LIN {X 0,Y 162.766,Z 348.566,A -85,B 0,C 180,E1 -23650.117,E2 -23650.117} C_VEL
LIN {X 0,Y 165.298,Z 338.62,A -85,B 0,C 180,E1 -23653.005,E2 -23653.005} C_VEL
LIN {X 0,Y 166.712,Z 332.788,A -85,B 0,C 180,E1 -23654.411,E2 -23654.411} C_VEL
LIN {X 0,Y 165.838,Z 322.83,A -85,B 0,C 180,E1 -23656.834,E2 -23656.834} C_VEL
LIN {X 0,Y 164.302,Z 311.523,A -85,B 0,C 180,E1 -23659.215,E2 -23659.215} C_VEL
LIN {X 0,Y 162.119,Z 300.27,A -85,B 0,C 180,E1 -23661.273,E2 -23661.273} C_VEL
LIN {X 0,Y 158.794,Z 286.809,A -85,B 0,C 180,E1 -23663.369,E2 -23663.369} C_VEL
LIN {X 0,Y 157.682,Z 283.839,A -85,B 0,C 180,E1 -23663.924,E2 -23663.924} C_VEL
LIN {X 0,Y 158.248,Z 283.771,A -85,B 0,C 180,E1 -23670,E2 -23670} C_VEL
LIN {X 0,Y 157.816,Z 283.83,A -85,B 0,C 180,E1 -23677.678,E2 -23677.678} C_VEL
LIN {X 0,Y 157.697,Z 283.837,A -85,B 0,C 180,E1 -23681.363,E2 -23681.363} C_VEL
LIN {X 0,Y 157.479,Z 283.868,A -85,B 0,C 180,E1 -23685.532,E2 -23685.532} C_VEL
LIN {X 0,Y 157.407,Z 283.876,A -85,B 0,C 180,E1 -23690.928,E2 -23690.928} C_VEL
LIN {X 0,Y 157.306,Z 283.879,A -85,B 0,C 180,E1 -23696.686,E2 -23696.686} C_VEL
LIN {X 0,Y 157.269,Z 283.893,A -85,B 0,C 180,E1 -23702.429,E2 -23702.429} C_VEL
LIN {X 0,Y 157.318,Z 283.886,A -85,B 0,C 180,E1 -23706.479,E2 -23706.479} C_VEL
LIN {X 0,Y 157.288,Z 283.866,A -85,B 0,C 180,E1 -23712.085,E2 -23712.085} C_VEL
LIN {X 0,Y 157.304,Z 283.881,A -85,B 0,C 180,E1 -23715.63,E2 -23715.63} C_VEL
LIN {X 0,Y 157.284,Z 283.893,A -85,B 0,C 180,E1 -23721.28,E2 -23721.28} C_VEL
LIN {X 0,Y 157.289,Z 283.885,A -85,B 0,C 180,E1 -23724.493,E2 -23724.493} C_VEL
LIN {X 0,Y 157.289,Z 283.864,A -85,B 0,C 180,E1 -23728.098,E2 -23728.098} C_VEL
LIN {X 0,Y 157.317,Z 283.878,A -85,B 0,C 180,E1 -23733.469,E2 -23733.469} C_VEL
LIN {X 0,Y 157.39,Z 283.878,A -85,B 0,C 180,E1 -23739.671,E2 -23739.671} C_VEL
LIN {X 0,Y 157.438,Z 283.857,A -85,B 0,C 180,E1 -23744.468,E2 -23744.468} C_VEL
LIN {X 0,Y 157.686,Z 283.82,A -85,B 0,C 180,E1 -23749.734,E2 -23749.734} C_VEL
LIN {X 0,Y 157.765,Z 283.822,A -85,B 0,C 180,E1 -23752.323,E2 -23752.323} C_VEL
LIN {X 0,Y 158.255,Z 283.768,A -85,B 0,C 180,E1 -23760.003,E2 -23760.003} C_VEL
LIN {X 0,Y 157.803,Z 283.815,A -85,B 0,C 180,E1 -23767.681,E2 -23767.681} C_VEL
LIN {X 0,Y 157.681,Z 283.842,A -85,B 0,C 180,E1 -23771.319,E2 -23771.319} C_VEL
LIN {X 0,Y 157.478,Z 283.864,A -85,B 0,C 180,E1 -23775.535,E2 -23775.535} C_VEL
LIN {X 0,Y 157.372,Z 283.876,A -85,B 0,C 180,E1 -23780.936,E2 -23780.936} C_VEL
LIN {X 0,Y 157.317,Z 283.884,A -85,B 0,C 180,E1 -23786.687,E2 -23786.687} C_VEL
LIN {X 0,Y 157.278,Z 283.896,A -85,B 0,C 180,E1 -23792.43,E2 -23792.43} C_VEL
LIN {X 0,Y 157.273,Z 283.892,A -85,B 0,C 180,E1 -23796.452,E2 -23796.452} C_VEL
LIN {X 0,Y 157.389,Z 283.892,A -85,B 0,C 180,E1 -23801.622,E2 -23801.622} C_VEL
LIN {X 0,Y 157.799,Z 286.274,A -85,B 0,C 180,E1 -23805.451,E2 -23805.451} C_VEL
LIN {X 0,Y 158.208,Z 288.611,A -85,B 0,C 180,E1 -23809.045,E2 -23809.045} C_VEL
LIN {X 0,Y 158.559,Z 290.868,A -85,B 0,C 180,E1 -23812.25,E2 -23812.25} C_VEL
LIN {X 0,Y 161.072,Z 302.499,A -85,B 0,C 180,E1 -23813.8,E2 -23813.8} C_VEL
LIN {X 0,Y 162.819,Z 314.796,A -85,B 0,C 180,E1 -23815.699,E2 -23815.699} C_VEL
LIN {X 0,Y 164.125,Z 327.048,A -85,B 0,C 180,E1 -23818.002,E2 -23818.002} C_VEL
LIN {X 0,Y 164.669,Z 338.78,A -85,B 0,C 180,E1 -23820.606,E2 -23820.606} C_VEL
LIN {X 0,Y 164.749,Z 346.799,A -85,B 0,C 180,E1 -23822.705,E2 -23822.705} C_VEL
LIN {X 0,Y 162.212,Z 356.942,A -85,B 0,C 180,E1 -23825.614,E2 -23825.614} C_VEL
LIN {X 0,Y 159.951,Z 365.602,A -85,B 0,C 180,E1 -23828.747,E2 -23828.747} C_VEL
LIN {X 0,Y 157.78,Z 373.82,A -85,B 0,C 180,E1 -23832.502,E2 -23832.502} C_VEL
LIN {X 0,Y 156.445,Z 379.436,A -85,B 0,C 180,E1 -23835.695,E2 -23835.695} C_VEL
LIN {X 0,Y 155.464,Z 384.917,A -85,B 0,C 180,E1 -23839.582,E2 -23839.582} C_VEL
LIN {X 0,Y 154.93,Z 389.177,A -85,B 0,C 180,E1 -23843.488,E2 -23843.488} C_VEL
LIN {X 0,Y 154.782,Z 392.343,A -85,B 0,C 180,E1 -23847.397,E2 -23847.397} C_VEL
LIN {X 0,Y 154.902,Z 393.899,A -85,B 0,C 180,E1 -23850,E2 -23850} C_VEL
LIN {X 0,Y 154.782,Z 395.024,A -85,B 0,C 180,E1 -23852.602,E2 -23852.602} C_VEL
LIN {X 0,Y 154.786,Z 395.727,A -85,B 0,C 180,E1 -23855.21,E2 -23855.21} C_VEL
LIN {X 0,Y 155.452,Z 395.975,A -85,B 0,C 180,E1 -23860.418,E2 -23860.418} C_VEL
LIN {X 0,Y 157.219,Z 394.762,A -85,B 0,C 180,E1 -23865.557,E2 -23865.557} C_VEL
LIN {X 0,Y 158.527,Z 393.574,A -85,B 0,C 180,E1 -23868.078,E2 -23868.078} C_VEL
LIN {X 0,Y 162.36,Z 390.018,A -85,B 0,C 180,E1 -23872.927,E2 -23872.927} C_VEL
LIN {X 0,Y 165.867,Z 386.263,A -85,B 0,C 180,E1 -23876.416,E2 -23876.416} C_VEL
LIN {X 0,Y 169.84,Z 381.521,A -85,B 0,C 180,E1 -23879.772,E2 -23879.772} C_VEL
LIN {X 0,Y 175.416,Z 374.551,A -85,B 0,C 180,E1 -23883.427,E2 -23883.427} C_VEL
LIN {X 0,Y 180.894,Z 367.066,A -85,B 0,C 180,E1 -23886.332,E2 -23886.332} C_VEL
LIN {X 0,Y 182.456,Z 364.28,A -85,B 0,C 180,E1 -23887.348,E2 -23887.348} C_VEL
LIN {X 0,Y 184.669,Z 357.993,A -85,B 0,C 180,E1 -23889.824,E2 -23889.824} C_VEL
LIN {X 0,Y 185.443,Z 355.091,A -85,B 0,C 180,E1 -23890.981,E2 -23890.981} C_VEL
LIN {X 0,Y 185.682,Z 351.795,A -85,B 0,C 180,E1 -23892.493,E2 -23892.493} C_VEL
LIN {X 0,Y 184.975,Z 349.138,A -85,B 0,C 180,E1 -23894.125,E2 -23894.125} C_VEL
LIN {X 0,Y 181.89,Z 343.339,A -85,B 0,C 180,E1 -23898.777,E2 -23898.777} C_VEL
LIN {X 0,Y 181.489,Z 341.7,A -85,B 0,C 180,E1 -23899.951,E2 -23899.951} C_VEL
LIN {X 0,Y 180.807,Z 337.52,A -85,B 0,C 180,E1 -23902.909,E2 -23902.909} C_VEL
LIN {X 0,Y 180.236,Z 335.055,A -85,B 0,C 180,E1 -23904.969,E2 -23904.969} C_VEL
LIN {X 0,Y 179.745,Z 332.311,A -85,B 0,C 180,E1 -23907.505,E2 -23907.505} C_VEL
LIN {X 0,Y 178.614,Z 327.494,A -85,B 0,C 180,E1 -23914.819,E2 -23914.819} C_VEL
LIN {X 0,Y 178.644,Z 326.719,A -85,B 0,C 180,E1 -23916.831,E2 -23916.831} C_VEL
LIN {X 0,Y 178.742,Z 326.277,A -85,B 0,C 180,E1 -23919.273,E2 -23919.273} C_VEL
LIN {X 0,Y 178.794,Z 326.661,A -85,B 0,C 180,E1 -23921.669,E2 -23921.669} C_VEL
LIN {X 0,Y 180.094,Z 329.764,A -85,B 0,C 180,E1 -23928.746,E2 -23928.746} C_VEL
LIN {X 0,Y 181.755,Z 335.002,A -85,B 0,C 180,E1 -23934.45,E2 -23934.45} C_VEL
LIN {X 0,Y 182.467,Z 339.478,A -85,B 0,C 180,E1 -23937.79,E2 -23937.79} C_VEL
LIN {X 0,Y 182.834,Z 344.048,A -85,B 0,C 180,E1 -23940.659,E2 -23940.659} C_VEL
LIN {X 0,Y 182.159,Z 350.277,A -85,B 0,C 180,E1 -23943.869,E2 -23943.869} C_VEL
LIN {X 0,Y 180.695,Z 356.16,A -85,B 0,C 180,E1 -23946.698,E2 -23946.698} C_VEL
LIN {X 0,Y 179.669,Z 358.308,A -85,B 0,C 180,E1 -23947.574,E2 -23947.574} C_VEL
LIN {X 0,Y 174.172,Z 365.633,A -85,B 0,C 180,E1 -23950.28,E2 -23950.28} C_VEL
LIN {X 0,Y 168.006,Z 372.913,A -85,B 0,C 180,E1 -23953.83,E2 -23953.83} C_VEL
LIN {X 0,Y 162.389,Z 378.767,A -85,B 0,C 180,E1 -23957.804,E2 -23957.804} C_VEL
LIN {X 0,Y 157.176,Z 383.446,A -85,B 0,C 180,E1 -23962.497,E2 -23962.497} C_VEL
LIN {X 0,Y 153.192,Z 386.436,A -85,B 0,C 180,E1 -23967.304,E2 -23967.304} C_VEL
LIN {X 0,Y 150.147,Z 387.993,A -85,B 0,C 180,E1 -23972.594,E2 -23972.594} C_VEL
LIN {X 0,Y 148.174,Z 388.041,A -85,B 0,C 180,E1 -23978.064,E2 -23978.064} C_VEL
LIN {X 0,Y 147.408,Z 387.123,A -85,B 0,C 180,E1 -23981.868,E2 -23981.868} C_VEL
LIN {X 0,Y 147.139,Z 385.428,A -85,B 0,C 180,E1 -23985.758,E2 -23985.758} C_VEL
LIN {X 0,Y 147.295,Z 382.83,A -85,B 0,C 180,E1 -23989.761,E2 -23989.761} C_VEL
LIN {X 0,Y 147.963,Z 379.18,A -85,B 0,C 180,E1 -23993.843,E2 -23993.843} C_VEL
LIN {X 0,Y 149.28,Z 373.176,A -85,B 0,C 180,E1 -23998.812,E2 -23998.812} C_VEL
LIN {X 0,Y 151.04,Z 366.254,A -85,B 0,C 180,E1 -24003.15,E2 -24003.15} C_VEL
LIN {X 0,Y 153.366,Z 357.835,A -85,B 0,C 180,E1 -24007.228,E2 -24007.228} C_VEL
LIN {X 0,Y 155.725,Z 349.243,A -85,B 0,C 180,E1 -24010.534,E2 -24010.534} C_VEL
LIN {X 0,Y 158.317,Z 339.375,A -85,B 0,C 180,E1 -24013.562,E2 -24013.562} C_VEL
LIN {X 0,Y 159.876,Z 332.712,A -85,B 0,C 180,E1 -24015.248,E2 -24015.248} C_VEL
LIN {X 0,Y 158.746,Z 321.108,A -85,B 0,C 180,E1 -24018.185,E2 -24018.185} C_VEL
LIN {X 0,Y 157.013,Z 309.073,A -85,B 0,C 180,E1 -24020.76,E2 -24020.76} C_VEL
LIN {X 0,Y 154.341,Z 296.343,A -85,B 0,C 180,E1 -24023.135,E2 -24023.135} C_VEL
LIN {X 0,Y 152.56,Z 289.599,A -85,B 0,C 180,E1 -24024.258,E2 -24024.258} C_VEL
LIN {X 0,Y 150.695,Z 285.026,A -85,B 0,C 180,E1 -24025.068,E2 -24025.068} C_VEL
LIN {X 0,Y 150.666,Z 284.718,A -85,B 0,C 180,E1 -24025.318,E2 -24025.318} C_VEL
LIN {X 0,Y 151.208,Z 284.648,A -85,B 0,C 180,E1 -24030,E2 -24030} C_VEL
LIN {X 0,Y 150.754,Z 284.71,A -85,B 0,C 180,E1 -24038.04,E2 -24038.04} C_VEL
LIN {X 0,Y 150.626,Z 284.718,A -85,B 0,C 180,E1 -24041.546,E2 -24041.546} C_VEL
LIN {X 0,Y 150.388,Z 284.747,A -85,B 0,C 180,E1 -24046.284,E2 -24046.284} C_VEL
LIN {X 0,Y 150.382,Z 284.751,A -85,B 0,C 180,E1 -24050.832,E2 -24050.832} C_VEL
LIN {X 0,Y 150.236,Z 284.755,A -85,B 0,C 180,E1 -24057.283,E2 -24057.283} C_VEL
LIN {X 0,Y 150.21,Z 284.773,A -85,B 0,C 180,E1 -24062.636,E2 -24062.636} C_VEL
LIN {X 0,Y 150.229,Z 284.766,A -85,B 0,C 180,E1 -24067.457,E2 -24067.457} C_VEL
LIN {X 0,Y 150.229,Z 284.745,A -85,B 0,C 180,E1 -24071.544,E2 -24071.544} C_VEL
LIN {X 0,Y 150.254,Z 284.757,A -85,B 0,C 180,E1 -24075.449,E2 -24075.449} C_VEL
LIN {X 0,Y 150.229,Z 284.771,A -85,B 0,C 180,E1 -24079.089,E2 -24079.089} C_VEL
LIN {X 0,Y 150.233,Z 284.769,A -85,B 0,C 180,E1 -24082.68,E2 -24082.68} C_VEL
LIN {X 0,Y 150.213,Z 284.748,A -85,B 0,C 180,E1 -24087.368,E2 -24087.368} C_VEL
LIN {X 0,Y 150.239,Z 284.754,A -85,B 0,C 180,E1 -24092.721,E2 -24092.721} C_VEL
LIN {X 0,Y 150.347,Z 284.756,A -85,B 0,C 180,E1 -24099.211,E2 -24099.211} C_VEL
LIN {X 0,Y 150.349,Z 284.745,A -85,B 0,C 180,E1 -24103.715,E2 -24103.715} C_VEL
LIN {X 0,Y 150.606,Z 284.696,A -85,B 0,C 180,E1 -24109.245,E2 -24109.245} C_VEL
LIN {X 0,Y 150.702,Z 284.7,A -85,B 0,C 180,E1 -24111.961,E2 -24111.961} C_VEL
LIN {X 0,Y 151.216,Z 284.644,A -85,B 0,C 180,E1 -24120.003,E2 -24120.003} C_VEL
LIN {X 0,Y 150.739,Z 284.696,A -85,B 0,C 180,E1 -24128.044,E2 -24128.044} C_VEL
LIN {X 0,Y 150.612,Z 284.723,A -85,B 0,C 180,E1 -24131.504,E2 -24131.504} C_VEL
LIN {X 0,Y 150.382,Z 284.743,A -85,B 0,C 180,E1 -24136.288,E2 -24136.288} C_VEL
LIN {X 0,Y 150.353,Z 284.75,A -85,B 0,C 180,E1 -24140.795,E2 -24140.795} C_VEL
LIN {X 0,Y 150.247,Z 284.762,A -85,B 0,C 180,E1 -24147.285,E2 -24147.285} C_VEL
LIN {X 0,Y 150.218,Z 284.776,A -85,B 0,C 180,E1 -24152.635,E2 -24152.635} C_VEL
LIN {X 0,Y 150.184,Z 284.779,A -85,B 0,C 180,E1 -24157.474,E2 -24157.474} C_VEL
LIN {X 0,Y 150.378,Z 284.841,A -85,B 0,C 180,E1 -24161.603,E2 -24161.603} C_VEL
LIN {X 0,Y 150.77,Z 287.258,A -85,B 0,C 180,E1 -24165.637,E2 -24165.637} C_VEL
LIN {X 0,Y 151.334,Z 290.659,A -85,B 0,C 180,E1 -24170.886,E2 -24170.886} C_VEL
LIN {X 0,Y 153.685,Z 298.998,A -85,B 0,C 180,E1 -24172.13,E2 -24172.13} C_VEL
LIN {X 0,Y 155.558,Z 311.145,A -85,B 0,C 180,E1 -24174.032,E2 -24174.032} C_VEL
LIN {X 0,Y 157.072,Z 324.55,A -85,B 0,C 180,E1 -24176.557,E2 -24176.557} C_VEL
LIN {X 0,Y 157.706,Z 335.061,A -85,B 0,C 180,E1 -24178.909,E2 -24178.909} C_VEL
LIN {X 0,Y 157.848,Z 345.901,A -85,B 0,C 180,E1 -24181.767,E2 -24181.767} C_VEL
LIN {X 0,Y 157.329,Z 349.398,A -85,B 0,C 180,E1 -24182.75,E2 -24182.75} C_VEL
LIN {X 0,Y 154.633,Z 359.142,A -85,B 0,C 180,E1 -24185.855,E2 -24185.855} C_VEL
LIN {X 0,Y 152.479,Z 367.199,A -85,B 0,C 180,E1 -24189.071,E2 -24189.071} C_VEL
LIN {X 0,Y 150.344,Z 375.101,A -85,B 0,C 180,E1 -24193.012,E2 -24193.012} C_VEL
LIN {X 0,Y 149.099,Z 380.453,A -85,B 0,C 180,E1 -24196.368,E2 -24196.368} C_VEL
LIN {X 0,Y 148.219,Z 385.687,A -85,B 0,C 180,E1 -24200.447,E2 -24200.447} C_VEL
LIN {X 0,Y 147.775,Z 389.713,A -85,B 0,C 180,E1 -24204.542,E2 -24204.542} C_VEL
LIN {X 0,Y 147.695,Z 392.183,A -85,B 0,C 180,E1 -24207.89,E2 -24207.89} C_VEL
LIN {X 0,Y 147.809,Z 393.41,A -85,B 0,C 180,E1 -24210,E2 -24210} C_VEL
LIN {X 0,Y 147.701,Z 394.601,A -85,B 0,C 180,E1 -24212.727,E2 -24212.727} C_VEL
LIN {X 0,Y 147.709,Z 395.398,A -85,B 0,C 180,E1 -24215.46,E2 -24215.46} C_VEL
LIN {X 0,Y 147.947,Z 395.797,A -85,B 0,C 180,E1 -24218.193,E2 -24218.193} C_VEL
LIN {X 0,Y 149.258,Z 395.448,A -85,B 0,C 180,E1 -24223.616,E2 -24223.616} C_VEL
LIN {X 0,Y 151.779,Z 393.647,A -85,B 0,C 180,E1 -24228.912,E2 -24228.912} C_VEL
LIN {X 0,Y 153.631,Z 392.168,A -85,B 0,C 180,E1 -24231.466,E2 -24231.466} C_VEL
LIN {X 0,Y 158.258,Z 387.996,A -85,B 0,C 180,E1 -24236.364,E2 -24236.364} C_VEL
LIN {X 0,Y 162.767,Z 383.216,A -85,B 0,C 180,E1 -24240.276,E2 -24240.276} C_VEL
LIN {X 0,Y 167.85,Z 377.486,A -85,B 0,C 180,E1 -24243.695,E2 -24243.695} C_VEL
LIN {X 0,Y 173.286,Z 370.738,A -85,B 0,C 180,E1 -24246.741,E2 -24246.741} C_VEL
LIN {X 0,Y 176.227,Z 366.828,A -85,B 0,C 180,E1 -24248.18,E2 -24248.18} C_VEL
LIN {X 0,Y 178.837,Z 360.757,A -85,B 0,C 180,E1 -24250.756,E2 -24250.756} C_VEL
LIN {X 0,Y 180.785,Z 353.995,A -85,B 0,C 180,E1 -24253.63,E2 -24253.63} C_VEL
LIN {X 0,Y 181.779,Z 348.847,A -85,B 0,C 180,E1 -24255.896,E2 -24255.896} C_VEL
LIN {X 0,Y 181.866,Z 345.381,A -85,B 0,C 180,E1 -24257.706,E2 -24257.706} C_VEL
LIN {X 0,Y 181.489,Z 341.7,A -85,B 0,C 180,E1 -24259.951,E2 -24259.951} C_VEL
LIN {X 0,Y 180.704,Z 339.737,A -85,B 0,C 180,E1 -24261.691,E2 -24261.691} C_VEL
LIN {X 0,Y 179.33,Z 338.667,A -85,B 0,C 180,E1 -24263.499,E2 -24263.499} C_VEL
LIN {X 0,Y 175.537,Z 337.281,A -85,B 0,C 180,E1 -24268.542,E2 -24268.542} C_VEL
LIN {X 0,Y 175.12,Z 336.621,A -85,B 0,C 180,E1 -24269.837,E2 -24269.837} C_VEL
LIN {X 0,Y 174.769,Z 334.192,A -85,B 0,C 180,E1 -24273.744,E2 -24273.744} C_VEL
LIN {X 0,Y 174.924,Z 332.649,A -85,B 0,C 180,E1 -24277.527,E2 -24277.527} C_VEL
LIN {X 0,Y 174.99,Z 332.407,A -85,B 0,C 180,E1 -24278.807,E2 -24278.807} C_VEL
LIN {X 0,Y 175.063,Z 332.617,A -85,B 0,C 180,E1 -24281.264,E2 -24281.264} C_VEL
LIN {X 0,Y 175.996,Z 335.511,A -85,B 0,C 180,E1 -24288.48,E2 -24288.48} C_VEL
LIN {X 0,Y 176.957,Z 339.379,A -85,B 0,C 180,E1 -24293.154,E2 -24293.154} C_VEL
LIN {X 0,Y 177.5,Z 343.407,A -85,B 0,C 180,E1 -24296.592,E2 -24296.592} C_VEL
LIN {X 0,Y 177.562,Z 348.314,A -85,B 0,C 180,E1 -24299.997,E2 -24299.997} C_VEL
LIN {X 0,Y 176.637,Z 353.41,A -85,B 0,C 180,E1 -24302.849,E2 -24302.849} C_VEL
LIN {X 0,Y 174.875,Z 359.006,A -85,B 0,C 180,E1 -24305.764,E2 -24305.764} C_VEL
LIN {X 0,Y 168.913,Z 366.651,A -85,B 0,C 180,E1 -24308.725,E2 -24308.725} C_VEL
LIN {X 0,Y 162.138,Z 374.054,A -85,B 0,C 180,E1 -24312.514,E2 -24312.514} C_VEL
LIN {X 0,Y 156.233,Z 379.619,A -85,B 0,C 180,E1 -24316.572,E2 -24316.572} C_VEL
LIN {X 0,Y 150.852,Z 384.044,A -85,B 0,C 180,E1 -24321.291,E2 -24321.291} C_VEL
LIN {X 0,Y 147.222,Z 386.501,A -85,B 0,C 180,E1 -24325.441,E2 -24325.441} C_VEL
LIN {X 0,Y 144.751,Z 387.774,A -85,B 0,C 180,E1 -24329.083,E2 -24329.083} C_VEL
LIN {X 0,Y 142.717,Z 388.396,A -85,B 0,C 180,E1 -24333.162,E2 -24333.162} C_VEL
LIN {X 0,Y 141.269,Z 388.228,A -85,B 0,C 180,E1 -24337.254,E2 -24337.254} C_VEL
LIN {X 0,Y 140.381,Z 387.25,A -85,B 0,C 180,E1 -24341.329,E2 -24341.329} C_VEL
LIN {X 0,Y 140.06,Z 385.51,A -85,B 0,C 180,E1 -24345.374,E2 -24345.374} C_VEL
LIN {X 0,Y 140.156,Z 383.054,A -85,B 0,C 180,E1 -24349.318,E2 -24349.318} C_VEL
LIN {X 0,Y 140.693,Z 379.862,A -85,B 0,C 180,E1 -24353.172,E2 -24353.172} C_VEL
LIN {X 0,Y 141.702,Z 375.212,A -85,B 0,C 180,E1 -24357.467,E2 -24357.467} C_VEL
LIN {X 0,Y 143.303,Z 368.887,A -85,B 0,C 180,E1 -24361.971,E2 -24361.971} C_VEL
LIN {X 0,Y 145.594,Z 360.66,A -85,B 0,C 180,E1 -24366.504,E2 -24366.504} C_VEL
LIN {X 0,Y 148.102,Z 351.955,A -85,B 0,C 180,E1 -24370.239,E2 -24370.239} C_VEL
LIN {X 0,Y 151.029,Z 341.386,A -85,B 0,C 180,E1 -24373.788,E2 -24373.788} C_VEL
LIN {X 0,Y 152.807,Z 334.817,A -85,B 0,C 180,E1 -24375.586,E2 -24375.586} C_VEL
LIN {X 0,Y 152.839,Z 330.773,A -85,B 0,C 180,E1 -24376.709,E2 -24376.709} C_VEL
LIN {X 0,Y 151.648,Z 319.16,A -85,B 0,C 180,E1 -24379.689,E2 -24379.689} C_VEL
LIN {X 0,Y 150.15,Z 309.08,A -85,B 0,C 180,E1 -24381.928,E2 -24381.928} C_VEL
LIN {X 0,Y 147.75,Z 297.311,A -85,B 0,C 180,E1 -24384.225,E2 -24384.225} C_VEL
LIN {X 0,Y 146.372,Z 292.363,A -85,B 0,C 180,E1 -24385.137,E2 -24385.137} C_VEL
LIN {X 0,Y 143.867,Z 286.452,A -85,B 0,C 180,E1 -24386.324,E2 -24386.324} C_VEL
LIN {X 0,Y 143.73,Z 285.58,A -85,B 0,C 180,E1 -24386.496,E2 -24386.496} C_VEL
LIN {X 0,Y 144.166,Z 285.525,A -85,B 0,C 180,E1 -24390,E2 -24390} C_VEL
LIN {X 0,Y 143.676,Z 285.59,A -85,B 0,C 180,E1 -24398.439,E2 -24398.439} C_VEL
LIN {X 0,Y 143.563,Z 285.599,A -85,B 0,C 180,E1 -24401.759,E2 -24401.759} C_VEL
LIN {X 0,Y 143.326,Z 285.623,A -85,B 0,C 180,E1 -24407.11,E2 -24407.11} C_VEL
LIN {X 0,Y 143.303,Z 285.633,A -85,B 0,C 180,E1 -24411.291,E2 -24411.291} C_VEL
LIN {X 0,Y 143.182,Z 285.632,A -85,B 0,C 180,E1 -24417.938,E2 -24417.938} C_VEL
LIN {X 0,Y 143.161,Z 285.652,A -85,B 0,C 180,E1 -24423.437,E2 -24423.437} C_VEL
LIN {X 0,Y 143.122,Z 285.639,A -85,B 0,C 180,E1 -24429.67,E2 -24429.67} C_VEL
LIN {X 0,Y 143.161,Z 285.628,A -85,B 0,C 180,E1 -24433.415,E2 -24433.415} C_VEL
LIN {X 0,Y 143.156,Z 285.649,A -85,B 0,C 180,E1 -24437.425,E2 -24437.425} C_VEL
LIN {X 0,Y 143.137,Z 285.653,A -85,B 0,C 180,E1 -24441.775,E2 -24441.775} C_VEL
LIN {X 0,Y 143.18,Z 285.623,A -85,B 0,C 180,E1 -24447.325,E2 -24447.325} C_VEL
LIN {X 0,Y 143.185,Z 285.63,A -85,B 0,C 180,E1 -24452.066,E2 -24452.066} C_VEL
LIN {X 0,Y 143.273,Z 285.639,A -85,B 0,C 180,E1 -24458.749,E2 -24458.749} C_VEL
LIN {X 0,Y 143.292,Z 285.625,A -85,B 0,C 180,E1 -24462.889,E2 -24462.889} C_VEL
LIN {X 0,Y 143.532,Z 285.572,A -85,B 0,C 180,E1 -24468.709,E2 -24468.709} C_VEL
LIN {X 0,Y 143.623,Z 285.581,A -85,B 0,C 180,E1 -24471.562,E2 -24471.562} C_VEL
LIN {X 0,Y 144.175,Z 285.521,A -85,B 0,C 180,E1 -24480.003,E2 -24480.003} C_VEL
LIN {X 0,Y 143.66,Z 285.58,A -85,B 0,C 180,E1 -24488.443,E2 -24488.443} C_VEL
LIN {X 0,Y 143.549,Z 285.604,A -85,B 0,C 180,E1 -24491.716,E2 -24491.716} C_VEL
LIN {X 0,Y 143.317,Z 285.619,A -85,B 0,C 180,E1 -24497.115,E2 -24497.115} C_VEL
LIN {X 0,Y 143.279,Z 285.632,A -85,B 0,C 180,E1 -24501.257,E2 -24501.257} C_VEL
LIN {X 0,Y 143.193,Z 285.639,A -85,B 0,C 180,E1 -24507.94,E2 -24507.94} C_VEL
LIN {X 0,Y 143.147,Z 285.656,A -85,B 0,C 180,E1 -24513.422,E2 -24513.422} C_VEL
LIN {X 0,Y 143.289,Z 285.635,A -85,B 0,C 180,E1 -24521.253,E2 -24521.253} C_VEL
LIN {X 0,Y 143.858,Z 288.991,A -85,B 0,C 180,E1 -24527.127,E2 -24527.127} C_VEL
LIN {X 0,Y 144.15,Z 290.566,A -85,B 0,C 180,E1 -24529.445,E2 -24529.445} C_VEL
LIN {X 0,Y 147.19,Z 300.178,A -85,B 0,C 180,E1 -24531.066,E2 -24531.066} C_VEL
LIN {X 0,Y 148.978,Z 312.003,A -85,B 0,C 180,E1 -24533.042,E2 -24533.042} C_VEL
LIN {X 0,Y 150.198,Z 323.899,A -85,B 0,C 180,E1 -24535.395,E2 -24535.395} C_VEL
LIN {X 0,Y 150.892,Z 335.228,A -85,B 0,C 180,E1 -24538.069,E2 -24538.069} C_VEL
LIN {X 0,Y 150.921,Z 346.18,A -85,B 0,C 180,E1 -24541.11,E2 -24541.11} C_VEL
LIN {X 0,Y 150.415,Z 349.648,A -85,B 0,C 180,E1 -24542.145,E2 -24542.145} C_VEL
LIN {X 0,Y 147.628,Z 359.316,A -85,B 0,C 180,E1 -24545.383,E2 -24545.383} C_VEL
LIN {X 0,Y 145.419,Z 367.313,A -85,B 0,C 180,E1 -24548.748,E2 -24548.748} C_VEL
LIN {X 0,Y 143.202,Z 375.144,A -85,B 0,C 180,E1 -24552.874,E2 -24552.874} C_VEL
LIN {X 0,Y 141.78,Z 381.408,A -85,B 0,C 180,E1 -24557.111,E2 -24557.111} C_VEL
LIN {X 0,Y 140.981,Z 386.372,A -85,B 0,C 180,E1 -24561.399,E2 -24561.399} C_VEL
LIN {X 0,Y 140.638,Z 390.162,A -85,B 0,C 180,E1 -24565.701,E2 -24565.701} C_VEL
LIN {X 0,Y 140.744,Z 392.908,A -85,B 0,C 180,E1 -24570,E2 -24570} C_VEL
LIN {X 0,Y 140.623,Z 394.158,A -85,B 0,C 180,E1 -24572.864,E2 -24572.864} C_VEL
LIN {X 0,Y 140.911,Z 395.511,A -85,B 0,C 180,E1 -24578.605,E2 -24578.605} C_VEL
LIN {X 0,Y 142.335,Z 395.346,A -85,B 0,C 180,E1 -24584.292,E2 -24584.292} C_VEL
LIN {X 0,Y 145.071,Z 393.696,A -85,B 0,C 180,E1 -24589.822,E2 -24589.822} C_VEL
LIN {X 0,Y 149.394,Z 390.566,A -85,B 0,C 180,E1 -24595.048,E2 -24595.048} C_VEL
LIN {X 0,Y 154.652,Z 385.768,A -85,B 0,C 180,E1 -24599.991,E2 -24599.991} C_VEL
LIN {X 0,Y 159.39,Z 381.026,A -85,B 0,C 180,E1 -24603.446,E2 -24603.446} C_VEL
LIN {X 0,Y 165.768,Z 374.09,A -85,B 0,C 180,E1 -24607.167,E2 -24607.167} C_VEL
LIN {X 0,Y 170.721,Z 368.002,A -85,B 0,C 180,E1 -24609.648,E2 -24609.648} C_VEL
LIN {X 0,Y 173.409,Z 362.294,A -85,B 0,C 180,E1 -24612.262,E2 -24612.262} C_VEL
LIN {X 0,Y 175.643,Z 355.816,A -85,B 0,C 180,E1 -24615.251,E2 -24615.251} C_VEL
LIN {X 0,Y 176.604,Z 351.399,A -85,B 0,C 180,E1 -24617.425,E2 -24617.425} C_VEL
LIN {X 0,Y 176.615,Z 346.603,A -85,B 0,C 180,E1 -24620.452,E2 -24620.452} C_VEL
LIN {X 0,Y 176.221,Z 342.879,A -85,B 0,C 180,E1 -24623.254,E2 -24623.254} C_VEL
LIN {X 0,Y 175.596,Z 338.669,A -85,B 0,C 180,E1 -24627.19,E2 -24627.19} C_VEL
LIN {X 0,Y 175.12,Z 336.621,A -85,B 0,C 180,E1 -24629.837,E2 -24629.837} C_VEL
LIN {X 0,Y 174.49,Z 335.988,A -85,B 0,C 180,E1 -24631.751,E2 -24631.751} C_VEL
LIN {X 0,Y 173.477,Z 336.228,A -85,B 0,C 180,E1 -24633.678,E2 -24633.678} C_VEL
LIN {X 0,Y 171.06,Z 338.221,A -85,B 0,C 180,E1 -24638.92,E2 -24638.92} C_VEL
LIN {X 0,Y 170.977,Z 338.405,A -85,B 0,C 180,E1 -24640.265,E2 -24640.265} C_VEL
LIN {X 0,Y 170.879,Z 339.238,A -85,B 0,C 180,E1 -24643.265,E2 -24643.265} C_VEL
LIN {X 0,Y 171.622,Z 341.068,A -85,B 0,C 180,E1 -24648.182,E2 -24648.182} C_VEL
LIN {X 0,Y 172.362,Z 345.483,A -85,B 0,C 180,E1 -24653.741,E2 -24653.741} C_VEL
LIN {X 0,Y 172.377,Z 350.164,A -85,B 0,C 180,E1 -24657.661,E2 -24657.661} C_VEL
LIN {X 0,Y 171.916,Z 353.532,A -85,B 0,C 180,E1 -24659.997,E2 -24659.997} C_VEL
LIN {X 0,Y 170.777,Z 357.511,A -85,B 0,C 180,E1 -24662.356,E2 -24662.356} C_VEL
LIN {X 0,Y 169.193,Z 361.369,A -85,B 0,C 180,E1 -24664.518,E2 -24664.518} C_VEL
LIN {X 0,Y 163.019,Z 368.528,A -85,B 0,C 180,E1 -24667.459,E2 -24667.459} C_VEL
LIN {X 0,Y 157.273,Z 374.326,A -85,B 0,C 180,E1 -24670.556,E2 -24670.556} C_VEL
LIN {X 0,Y 152.045,Z 379.02,A -85,B 0,C 180,E1 -24673.914,E2 -24673.914} C_VEL
LIN {X 0,Y 147.357,Z 382.688,A -85,B 0,C 180,E1 -24677.474,E2 -24677.474} C_VEL
LIN {X 0,Y 143.312,Z 385.434,A -85,B 0,C 180,E1 -24681.294,E2 -24681.294} C_VEL
LIN {X 0,Y 139.935,Z 387.327,A -85,B 0,C 180,E1 -24685.311,E2 -24685.311} C_VEL
LIN {X 0,Y 136.47,Z 388.588,A -85,B 0,C 180,E1 -24690.992,E2 -24690.992} C_VEL
LIN {X 0,Y 134.825,Z 388.551,A -85,B 0,C 180,E1 -24694.983,E2 -24694.983} C_VEL
LIN {X 0,Y 133.665,Z 387.833,A -85,B 0,C 180,E1 -24699.115,E2 -24699.115} C_VEL
LIN {X 0,Y 133.038,Z 386.364,A -85,B 0,C 180,E1 -24703.368,E2 -24703.368} C_VEL
LIN {X 0,Y 133.049,Z 382.992,A -85,B 0,C 180,E1 -24709.219,E2 -24709.219} C_VEL
LIN {X 0,Y 133.913,Z 378.311,A -85,B 0,C 180,E1 -24714.741,E2 -24714.741} C_VEL
LIN {X 0,Y 135.169,Z 373.002,A -85,B 0,C 180,E1 -24719.389,E2 -24719.389} C_VEL
LIN {X 0,Y 137.105,Z 365.888,A -85,B 0,C 180,E1 -24724.171,E2 -24724.171} C_VEL
LIN {X 0,Y 139.604,Z 357.427,A -85,B 0,C 180,E1 -24728.594,E2 -24728.594} C_VEL
LIN {X 0,Y 142.351,Z 348.218,A -85,B 0,C 180,E1 -24732.358,E2 -24732.358} C_VEL
LIN {X 0,Y 145.15,Z 338.325,A -85,B 0,C 180,E1 -24735.537,E2 -24735.537} C_VEL
LIN {X 0,Y 146.053,Z 335.084,A -85,B 0,C 180,E1 -24736.434,E2 -24736.434} C_VEL
LIN {X 0,Y 145.666,Z 327.893,A -85,B 0,C 180,E1 -24738.521,E2 -24738.521} C_VEL
LIN {X 0,Y 144.618,Z 317.674,A -85,B 0,C 180,E1 -24741.18,E2 -24741.18} C_VEL
LIN {X 0,Y 142.726,Z 305.812,A -85,B 0,C 180,E1 -24743.888,E2 -24743.888} C_VEL
LIN {X 0,Y 140.688,Z 296.26,A -85,B 0,C 180,E1 -24745.827,E2 -24745.827} C_VEL
LIN {X 0,Y 136.967,Z 287.334,A -85,B 0,C 180,E1 -24747.795,E2 -24747.795} C_VEL
LIN {X 0,Y 136.815,Z 286.442,A -85,B 0,C 180,E1 -24747.977,E2 -24747.977} C_VEL
LIN {X 0,Y 137.122,Z 286.402,A -85,B 0,C 180,E1 -24750,E2 -24750} C_VEL
LIN {X 0,Y 136.6,Z 286.47,A -85,B 0,C 180,E1 -24758.879,E2 -24758.879} C_VEL
LIN {X 0,Y 136.485,Z 286.481,A -85,B 0,C 180,E1 -24761.96,E2 -24761.96} C_VEL
LIN {X 0,Y 136.265,Z 286.5,A -85,B 0,C 180,E1 -24768.026,E2 -24768.026} C_VEL
LIN {X 0,Y 136.219,Z 286.517,A -85,B 0,C 180,E1 -24771.781,E2 -24771.781} C_VEL
LIN {X 0,Y 136.092,Z 286.515,A -85,B 0,C 180,E1 -24778.618,E2 -24778.618} C_VEL
LIN {X 0,Y 136.075,Z 286.535,A -85,B 0,C 180,E1 -24784.619,E2 -24784.619} C_VEL
LIN {X 0,Y 136.096,Z 286.516,A -85,B 0,C 180,E1 -24789.238,E2 -24789.238} C_VEL
LIN {X 0,Y 136.097,Z 286.509,A -85,B 0,C 180,E1 -24793.707,E2 -24793.707} C_VEL
LIN {X 0,Y 136.104,Z 286.53,A -85,B 0,C 180,E1 -24797.839,E2 -24797.839} C_VEL
LIN {X 0,Y 136.089,Z 286.531,A -85,B 0,C 180,E1 -24801.71,E2 -24801.71} C_VEL
LIN {X 0,Y 136.087,Z 286.517,A -85,B 0,C 180,E1 -24805.719,E2 -24805.719} C_VEL
LIN {X 0,Y 136.142,Z 286.507,A -85,B 0,C 180,E1 -24812.32,E2 -24812.32} C_VEL
LIN {X 0,Y 136.24,Z 286.515,A -85,B 0,C 180,E1 -24818.836,E2 -24818.836} C_VEL
LIN {X 0,Y 136.258,Z 286.49,A -85,B 0,C 180,E1 -24825.059,E2 -24825.059} C_VEL
LIN {X 0,Y 136.425,Z 286.454,A -85,B 0,C 180,E1 -24828.176,E2 -24828.176} C_VEL
LIN {X 0,Y 136.548,Z 286.457,A -85,B 0,C 180,E1 -24831.121,E2 -24831.121} C_VEL
LIN {X 0,Y 137.132,Z 286.398,A -85,B 0,C 180,E1 -24840.003,E2 -24840.003} C_VEL
LIN {X 0,Y 136.588,Z 286.464,A -85,B 0,C 180,E1 -24848.883,E2 -24848.883} C_VEL
LIN {X 0,Y 136.492,Z 286.484,A -85,B 0,C 180,E1 -24851.958,E2 -24851.958} C_VEL
LIN {X 0,Y 136.253,Z 286.495,A -85,B 0,C 180,E1 -24858.032,E2 -24858.032} C_VEL
LIN {X 0,Y 136.2,Z 286.516,A -85,B 0,C 180,E1 -24861.752,E2 -24861.752} C_VEL
LIN {X 0,Y 136.103,Z 286.523,A -85,B 0,C 180,E1 -24868.619,E2 -24868.619} C_VEL
LIN {X 0,Y 136.047,Z 286.536,A -85,B 0,C 180,E1 -24874.632,E2 -24874.632} C_VEL
LIN {X 0,Y 136.246,Z 286.574,A -85,B 0,C 180,E1 -24881.301,E2 -24881.301} C_VEL
LIN {X 0,Y 136.803,Z 289.663,A -85,B 0,C 180,E1 -24886.957,E2 -24886.957} C_VEL
LIN {X 0,Y 136.873,Z 290.167,A -85,B 0,C 180,E1 -24887.78,E2 -24887.78} C_VEL
LIN {X 0,Y 137.884,Z 293.393,A -85,B 0,C 180,E1 -24888.34,E2 -24888.34} C_VEL
LIN {X 0,Y 140.858,Z 302.164,A -85,B 0,C 180,E1 -24890.049,E2 -24890.049} C_VEL
LIN {X 0,Y 142.461,Z 313.551,A -85,B 0,C 180,E1 -24892.127,E2 -24892.127} C_VEL
LIN {X 0,Y 143.559,Z 325.762,A -85,B 0,C 180,E1 -24894.75,E2 -24894.75} C_VEL
LIN {X 0,Y 144.054,Z 335.366,A -85,B 0,C 180,E1 -24897.156,E2 -24897.156} C_VEL
LIN {X 0,Y 144.05,Z 346.456,A -85,B 0,C 180,E1 -24900.397,E2 -24900.397} C_VEL
LIN {X 0,Y 143.569,Z 349.714,A -85,B 0,C 180,E1 -24901.426,E2 -24901.426} C_VEL
LIN {X 0,Y 140.656,Z 359.466,A -85,B 0,C 180,E1 -24904.868,E2 -24904.868} C_VEL
LIN {X 0,Y 138.353,Z 367.383,A -85,B 0,C 180,E1 -24908.39,E2 -24908.39} C_VEL
LIN {X 0,Y 136.094,Z 375.133,A -85,B 0,C 180,E1 -24912.726,E2 -24912.726} C_VEL
LIN {X 0,Y 134.483,Z 382.243,A -85,B 0,C 180,E1 -24917.934,E2 -24917.934} C_VEL
LIN {X 0,Y 133.77,Z 386.963,A -85,B 0,C 180,E1 -24922.452,E2 -24922.452} C_VEL
LIN {X 0,Y 133.564,Z 390.54,A -85,B 0,C 180,E1 -24926.983,E2 -24926.983} C_VEL
LIN {X 0,Y 133.668,Z 392.366,A -85,B 0,C 180,E1 -24930,E2 -24930} C_VEL
LIN {X 0,Y 133.56,Z 393.713,A -85,B 0,C 180,E1 -24933.016,E2 -24933.016} C_VEL
LIN {X 0,Y 133.875,Z 395.202,A -85,B 0,C 180,E1 -24939.061,E2 -24939.061} C_VEL
LIN {X 0,Y 135.442,Z 395.229,A -85,B 0,C 180,E1 -24945.036,E2 -24945.036} C_VEL
LIN {X 0,Y 138.409,Z 393.755,A -85,B 0,C 180,E1 -24950.82,E2 -24950.82} C_VEL
LIN {X 0,Y 142.983,Z 390.79,A -85,B 0,C 180,E1 -24956.254,E2 -24956.254} C_VEL
LIN {X 0,Y 147.075,Z 387.538,A -85,B 0,C 180,E1 -24960.114,E2 -24960.114} C_VEL
LIN {X 0,Y 151.798,Z 383.344,A -85,B 0,C 180,E1 -24963.75,E2 -24963.75} C_VEL
LIN {X 0,Y 157.324,Z 378.071,A -85,B 0,C 180,E1 -24967.089,E2 -24967.089} C_VEL
LIN {X 0,Y 163.335,Z 371.588,A -85,B 0,C 180,E1 -24970.196,E2 -24970.196} C_VEL
LIN {X 0,Y 165.317,Z 369.156,A -85,B 0,C 180,E1 -24971.218,E2 -24971.218} C_VEL
LIN {X 0,Y 167.689,Z 364.783,A -85,B 0,C 180,E1 -24973.39,E2 -24973.39} C_VEL
LIN {X 0,Y 170.128,Z 358.98,A -85,B 0,C 180,E1 -24976.293,E2 -24976.293} C_VEL
LIN {X 0,Y 171.273,Z 354.904,A -85,B 0,C 180,E1 -24978.482,E2 -24978.482} C_VEL
LIN {X 0,Y 171.529,Z 351.092,A -85,B 0,C 180,E1 -24981.12,E2 -24981.12} C_VEL
LIN {X 0,Y 171.326,Z 346.387,A -85,B 0,C 180,E1 -24985.125,E2 -24985.125} C_VEL
LIN {X 0,Y 171.087,Z 343.924,A -85,B 0,C 180,E1 -24987.72,E2 -24987.72} C_VEL
LIN {X 0,Y 170.786,Z 342.007,A -85,B 0,C 180,E1 -24990.406,E2 -24990.406} C_VEL
LIN {X 0,Y 170.773,Z 339.167,A -85,B 0,C 180,E1 -24995.696,E2 -24995.696} C_VEL
LIN {X 0,Y 170.941,Z 338.37,A -85,B 0,C 180,E1 -24998.28,E2 -24998.28} C_VEL
LIN {X 0,Y 170.977,Z 338.405,A -85,B 0,C 180,E1 -25000.265,E2 -25000.265} C_VEL
LIN {X 0,Y 170.726,Z 339.137,A -85,B 0,C 180,E1 -25002.217,E2 -25002.217} C_VEL
LIN {X 0,Y 169.903,Z 340.879,A -85,B 0,C 180,E1 -25004.103,E2 -25004.103} C_VEL
LIN {X 0,Y 167.24,Z 347.008,A -85,B 0,C 180,E1 -25009.101,E2 -25009.101} C_VEL
LIN {X 0,Y 167.093,Z 348.172,A -85,B 0,C 180,E1 -25010.426,E2 -25010.426} C_VEL
LIN {X 0,Y 167.35,Z 349.867,A -85,B 0,C 180,E1 -25012.759,E2 -25012.759} C_VEL
LIN {X 0,Y 167.106,Z 353.661,A -85,B 0,C 180,E1 -25016.38,E2 -25016.38} C_VEL
LIN {X 0,Y 166.526,Z 356.712,A -85,B 0,C 180,E1 -25018.788,E2 -25018.788} C_VEL
LIN {X 0,Y 165.214,Z 360.383,A -85,B 0,C 180,E1 -25021.216,E2 -25021.216} C_VEL
LIN {X 0,Y 163.665,Z 363.559,A -85,B 0,C 180,E1 -25023.139,E2 -25023.139} C_VEL
LIN {X 0,Y 157.509,Z 370.028,A -85,B 0,C 180,E1 -25025.936,E2 -25025.936} C_VEL
LIN {X 0,Y 151.749,Z 375.348,A -85,B 0,C 180,E1 -25028.955,E2 -25028.955} C_VEL
LIN {X 0,Y 144.565,Z 381.133,A -85,B 0,C 180,E1 -25033.525,E2 -25033.525} C_VEL
LIN {X 0,Y 139.498,Z 384.573,A -85,B 0,C 180,E1 -25037.591,E2 -25037.591} C_VEL
LIN {X 0,Y 135.773,Z 386.666,A -85,B 0,C 180,E1 -25041.298,E2 -25041.298} C_VEL
LIN {X 0,Y 132.391,Z 388.149,A -85,B 0,C 180,E1 -25045.521,E2 -25045.521} C_VEL
LIN {X 0,Y 129.744,Z 388.833,A -85,B 0,C 180,E1 -25049.926,E2 -25049.926} C_VEL
LIN {X 0,Y 127.833,Z 388.711,A -85,B 0,C 180,E1 -25054.448,E2 -25054.448} C_VEL
LIN {X 0,Y 126.561,Z 387.779,A -85,B 0,C 180,E1 -25058.977,E2 -25058.977} C_VEL
LIN {X 0,Y 125.925,Z 386.107,A -85,B 0,C 180,E1 -25063.488,E2 -25063.488} C_VEL
LIN {X 0,Y 125.89,Z 383.7,A -85,B 0,C 180,E1 -25067.941,E2 -25067.941} C_VEL
LIN {X 0,Y 126.302,Z 380.549,A -85,B 0,C 180,E1 -25072.261,E2 -25072.261} C_VEL
LIN {X 0,Y 127.473,Z 375.501,A -85,B 0,C 180,E1 -25077.484,E2 -25077.484} C_VEL
LIN {X 0,Y 129.226,Z 368.839,A -85,B 0,C 180,E1 -25082.69,E2 -25082.69} C_VEL
LIN {X 0,Y 131.359,Z 361.671,A -85,B 0,C 180,E1 -25087.068,E2 -25087.068} C_VEL
LIN {X 0,Y 133.824,Z 353.692,A -85,B 0,C 180,E1 -25090.949,E2 -25090.949} C_VEL
LIN {X 0,Y 136.824,Z 343.808,A -85,B 0,C 180,E1 -25094.738,E2 -25094.738} C_VEL
LIN {X 0,Y 139.249,Z 335.637,A -85,B 0,C 180,E1 -25097.244,E2 -25097.244} C_VEL
LIN {X 0,Y 138.687,Z 326.08,A -85,B 0,C 180,E1 -25100.153,E2 -25100.153} C_VEL
LIN {X 0,Y 137.491,Z 315.008,A -85,B 0,C 180,E1 -25103.096,E2 -25103.096} C_VEL
LIN {X 0,Y 135.3,Z 302.523,A -85,B 0,C 180,E1 -25106.03,E2 -25106.03} C_VEL
LIN {X 0,Y 134.671,Z 299.452,A -85,B 0,C 180,E1 -25106.677,E2 -25106.677} C_VEL
LIN {X 0,Y 130.124,Z 288.164,A -85,B 0,C 180,E1 -25109.362,E2 -25109.362} C_VEL
LIN {X 0,Y 129.997,Z 287.291,A -85,B 0,C 180,E1 -25109.575,E2 -25109.575} C_VEL
LIN {X 0,Y 129.506,Z 287.354,A -85,B 0,C 180,E1 -25116.231,E2 -25116.231} C_VEL
LIN {X 0,Y 129.522,Z 287.35,A -85,B 0,C 180,E1 -25119.369,E2 -25119.369} C_VEL
LIN {X 0,Y 129.387,Z 287.368,A -85,B 0,C 180,E1 -25122.549,E2 -25122.549} C_VEL
LIN {X 0,Y 129.177,Z 287.386,A -85,B 0,C 180,E1 -25129.053,E2 -25129.053} C_VEL
LIN {X 0,Y 129.128,Z 287.401,A -85,B 0,C 180,E1 -25132.395,E2 -25132.395} C_VEL
LIN {X 0,Y 129.009,Z 287.399,A -85,B 0,C 180,E1 -25139.36,E2 -25139.36} C_VEL
LIN {X 0,Y 129.02,Z 287.414,A -85,B 0,C 180,E1 -25145.214,E2 -25145.214} C_VEL
LIN {X 0,Y 129.04,Z 287.383,A -85,B 0,C 180,E1 -25150.811,E2 -25150.811} C_VEL
LIN {X 0,Y 129.021,Z 287.398,A -85,B 0,C 180,E1 -25155.083,E2 -25155.083} C_VEL
LIN {X 0,Y 129.011,Z 287.415,A -85,B 0,C 180,E1 -25159.699,E2 -25159.699} C_VEL
LIN {X 0,Y 129.02,Z 287.4,A -85,B 0,C 180,E1 -25164.793,E2 -25164.793} C_VEL
LIN {X 0,Y 129.011,Z 287.382,A -85,B 0,C 180,E1 -25170.645,E2 -25170.645} C_VEL
LIN {X 0,Y 129.026,Z 287.403,A -85,B 0,C 180,E1 -25174.171,E2 -25174.171} C_VEL
LIN {X 0,Y 129.104,Z 287.402,A -85,B 0,C 180,E1 -25177.731,E2 -25177.731} C_VEL
LIN {X 0,Y 129.147,Z 287.394,A -85,B 0,C 180,E1 -25180.947,E2 -25180.947} C_VEL
LIN {X 0,Y 129.349,Z 287.334,A -85,B 0,C 180,E1 -25187.958,E2 -25187.958} C_VEL
LIN {X 0,Y 129.47,Z 287.334,A -85,B 0,C 180,E1 -25190.632,E2 -25190.632} C_VEL
LIN {X 0,Y 130.087,Z 287.275,A -85,B 0,C 180,E1 -25200.004,E2 -25200.004} C_VEL
LIN {X 0,Y 129.515,Z 287.346,A -85,B 0,C 180,E1 -25209.373,E2 -25209.373} C_VEL
LIN {X 0,Y 129.395,Z 287.367,A -85,B 0,C 180,E1 -25212.552,E2 -25212.552} C_VEL
LIN {X 0,Y 129.161,Z 287.378,A -85,B 0,C 180,E1 -25219.059,E2 -25219.059} C_VEL
LIN {X 0,Y 129.111,Z 287.401,A -85,B 0,C 180,E1 -25222.402,E2 -25222.402} C_VEL
LIN {X 0,Y 129.033,Z 287.408,A -85,B 0,C 180,E1 -25225.836,E2 -25225.836} C_VEL
LIN {X 0,Y 129.02,Z 287.408,A -85,B 0,C 180,E1 -25229.361,E2 -25229.361} C_VEL
LIN {X 0,Y 128.969,Z 287.416,A -85,B 0,C 180,E1 -25235.175,E2 -25235.175} C_VEL
LIN {X 0,Y 129.211,Z 287.486,A -85,B 0,C 180,E1 -25241.266,E2 -25241.266} C_VEL
LIN {X 0,Y 129.653,Z 289.941,A -85,B 0,C 180,E1 -25246.005,E2 -25246.005} C_VEL
LIN {X 0,Y 130.641,Z 293.103,A -85,B 0,C 180,E1 -25246.592,E2 -25246.592} C_VEL
LIN {X 0,Y 133.793,Z 301.706,A -85,B 0,C 180,E1 -25248.433,E2 -25248.433} C_VEL
LIN {X 0,Y 134.955,Z 306.628,A -85,B 0,C 180,E1 -25249.441,E2 -25249.441} C_VEL
LIN {X 0,Y 136.212,Z 317.85,A -85,B 0,C 180,E1 -25251.746,E2 -25251.746} C_VEL
LIN {X 0,Y 137.051,Z 329.526,A -85,B 0,C 180,E1 -25254.556,E2 -25254.556} C_VEL
LIN {X 0,Y 137.286,Z 338.49,A -85,B 0,C 180,E1 -25257.049,E2 -25257.049} C_VEL
LIN {X 0,Y 137.106,Z 347.79,A -85,B 0,C 180,E1 -25260.016,E2 -25260.016} C_VEL
LIN {X 0,Y 134.804,Z 355.929,A -85,B 0,C 180,E1 -25262.859,E2 -25262.859} C_VEL
LIN {X 0,Y 132.207,Z 364.422,A -85,B 0,C 180,E1 -25266.503,E2 -25266.503} C_VEL
LIN {X 0,Y 129.674,Z 372.678,A -85,B 0,C 180,E1 -25271.023,E2 -25271.023} C_VEL
LIN {X 0,Y 127.922,Z 379.341,A -85,B 0,C 180,E1 -25275.686,E2 -25275.686} C_VEL
LIN {X 0,Y 126.947,Z 384.655,A -85,B 0,C 180,E1 -25280.439,E2 -25280.439} C_VEL
LIN {X 0,Y 126.517,Z 388.758,A -85,B 0,C 180,E1 -25285.22,E2 -25285.22} C_VEL
LIN {X 0,Y 126.6,Z 391.78,A -85,B 0,C 180,E1 -25290,E2 -25290} C_VEL
LIN {X 0,Y 126.492,Z 393.222,A -85,B 0,C 180,E1 -25293.185,E2 -25293.185} C_VEL
LIN {X 0,Y 126.51,Z 394.253,A -85,B 0,C 180,E1 -25296.378,E2 -25296.378} C_VEL
LIN {X 0,Y 127.55,Z 395.152,A -85,B 0,C 180,E1 -25302.732,E2 -25302.732} C_VEL
LIN {X 0,Y 129.947,Z 394.616,A -85,B 0,C 180,E1 -25308.934,E2 -25308.934} C_VEL
LIN {X 0,Y 134.043,Z 392.611,A -85,B 0,C 180,E1 -25314.799,E2 -25314.799} C_VEL
LIN {X 0,Y 139.47,Z 389.085,A -85,B 0,C 180,E1 -25320.258,E2 -25320.258} C_VEL
LIN {X 0,Y 144.174,Z 385.44,A -85,B 0,C 180,E1 -25324.03,E2 -25324.03} C_VEL
LIN {X 0,Y 149.75,Z 380.678,A -85,B 0,C 180,E1 -25327.596,E2 -25327.596} C_VEL
LIN {X 0,Y 156.909,Z 373.822,A -85,B 0,C 180,E1 -25331.348,E2 -25331.348} C_VEL
LIN {X 0,Y 159.166,Z 371.51,A -85,B 0,C 180,E1 -25332.326,E2 -25332.326} C_VEL
LIN {X 0,Y 161.508,Z 368.045,A -85,B 0,C 180,E1 -25334.124,E2 -25334.124} C_VEL
LIN {X 0,Y 164.609,Z 361.92,A -85,B 0,C 180,E1 -25337.432,E2 -25337.432} C_VEL
LIN {X 0,Y 165.613,Z 359.404,A -85,B 0,C 180,E1 -25338.87,E2 -25338.87} C_VEL
LIN {X 0,Y 166.124,Z 356.905,A -85,B 0,C 180,E1 -25340.608,E2 -25340.608} C_VEL
LIN {X 0,Y 166.342,Z 353.226,A -85,B 0,C 180,E1 -25343.733,E2 -25343.733} C_VEL
LIN {X 0,Y 166.366,Z 349.484,A -85,B 0,C 180,E1 -25347.657,E2 -25347.657} C_VEL
LIN {X 0,Y 166.273,Z 348.108,A -85,B 0,C 180,E1 -25349.519,E2 -25349.519} C_VEL
LIN {X 0,Y 166.31,Z 345.147,A -85,B 0,C 180,E1 -25354.999,E2 -25354.999} C_VEL
LIN {X 0,Y 166.608,Z 344.093,A -85,B 0,C 180,E1 -25358.125,E2 -25358.125} C_VEL
LIN {X 0,Y 166.668,Z 344.047,A -85,B 0,C 180,E1 -25360.282,E2 -25360.282} C_VEL
LIN {X 0,Y 166.997,Z 346.411,A -85,B 0,C 180,E1 -25367.85,E2 -25367.85} C_VEL
LIN {X 0,Y 167.093,Z 348.172,A -85,B 0,C 180,E1 -25370.426,E2 -25370.426} C_VEL
LIN {X 0,Y 166.908,Z 349.423,A -85,B 0,C 180,E1 -25371.714,E2 -25371.714} C_VEL
LIN {X 0,Y 166.31,Z 351.104,A -85,B 0,C 180,E1 -25372.935,E2 -25372.935} C_VEL
LIN {X 0,Y 164.297,Z 355.095,A -85,B 0,C 180,E1 -25375.238,E2 -25375.238} C_VEL
LIN {X 0,Y 161.802,Z 359.339,A -85,B 0,C 180,E1 -25377.527,E2 -25377.527} C_VEL
LIN {X 0,Y 159.691,Z 363.15,A -85,B 0,C 180,E1 -25379.964,E2 -25379.964} C_VEL
LIN {X 0,Y 158.653,Z 365.042,A -85,B 0,C 180,E1 -25381.266,E2 -25381.266} C_VEL
LIN {X 0,Y 155.924,Z 367.944,A -85,B 0,C 180,E1 -25382.58,E2 -25382.58} C_VEL
LIN {X 0,Y 148.438,Z 374.768,A -85,B 0,C 180,E1 -25386.15,E2 -25386.15} C_VEL
LIN {X 0,Y 140.999,Z 380.445,A -85,B 0,C 180,E1 -25390.435,E2 -25390.435} C_VEL
LIN {X 0,Y 134.519,Z 384.586,A -85,B 0,C 180,E1 -25395.139,E2 -25395.139} C_VEL
LIN {X 0,Y 130.468,Z 386.719,A -85,B 0,C 180,E1 -25398.853,E2 -25398.853} C_VEL
LIN {X 0,Y 126.976,Z 388.192,A -85,B 0,C 180,E1 -25402.791,E2 -25402.791} C_VEL
LIN {X 0,Y 124.121,Z 388.948,A -85,B 0,C 180,E1 -25406.93,E2 -25406.93} C_VEL
LIN {X 0,Y 121.892,Z 389.052,A -85,B 0,C 180,E1 -25411.255,E2 -25411.255} C_VEL
LIN {X 0,Y 120.222,Z 388.49,A -85,B 0,C 180,E1 -25415.768,E2 -25415.768} C_VEL
LIN {X 0,Y 119.165,Z 387.147,A -85,B 0,C 180,E1 -25420.441,E2 -25420.441} C_VEL
LIN {X 0,Y 118.764,Z 385.026,A -85,B 0,C 180,E1 -25425.238,E2 -25425.238} C_VEL
LIN {X 0,Y 118.949,Z 381.982,A -85,B 0,C 180,E1 -25430.176,E2 -25430.176} C_VEL
LIN {X 0,Y 119.779,Z 377.839,A -85,B 0,C 180,E1 -25435.222,E2 -25435.222} C_VEL
LIN {X 0,Y 121.188,Z 372.251,A -85,B 0,C 180,E1 -25440.436,E2 -25440.436} C_VEL
LIN {X 0,Y 123.346,Z 364.923,A -85,B 0,C 180,E1 -25445.724,E2 -25445.724} C_VEL
LIN {X 0,Y 126.112,Z 356.394,A -85,B 0,C 180,E1 -25450.467,E2 -25450.467} C_VEL
LIN {X 0,Y 129.25,Z 346.556,A -85,B 0,C 180,E1 -25454.686,E2 -25454.686} C_VEL
LIN {X 0,Y 132.451,Z 336.198,A -85,B 0,C 180,E1 -25458.135,E2 -25458.135} C_VEL
LIN {X 0,Y 131.841,Z 325.48,A -85,B 0,C 180,E1 -25461.571,E2 -25461.571} C_VEL
LIN {X 0,Y 130.718,Z 314.879,A -85,B 0,C 180,E1 -25464.517,E2 -25464.517} C_VEL
LIN {X 0,Y 128.488,Z 302.267,A -85,B 0,C 180,E1 -25467.65,E2 -25467.65} C_VEL
LIN {X 0,Y 123.968,Z 291.086,A -85,B 0,C 180,E1 -25470.66,E2 -25470.66} C_VEL
LIN {X 0,Y 122.813,Z 288.186,A -85,B 0,C 180,E1 -25471.435,E2 -25471.435} C_VEL
LIN {X 0,Y 122.449,Z 288.228,A -85,B 0,C 180,E1 -25479.915,E2 -25479.915} C_VEL
LIN {X 0,Y 122.28,Z 288.254,A -85,B 0,C 180,E1 -25483.291,E2 -25483.291} C_VEL
LIN {X 0,Y 122.065,Z 288.275,A -85,B 0,C 180,E1 -25490.21,E2 -25490.21} C_VEL
LIN {X 0,Y 121.988,Z 288.288,A -85,B 0,C 180,E1 -25493.784,E2 -25493.784} C_VEL
LIN {X 0,Y 121.922,Z 288.285,A -85,B 0,C 180,E1 -25500.166,E2 -25500.166} C_VEL
LIN {X 0,Y 121.96,Z 288.29,A -85,B 0,C 180,E1 -25506.227,E2 -25506.227} C_VEL
LIN {X 0,Y 121.959,Z 288.262,A -85,B 0,C 180,E1 -25511.491,E2 -25511.491} C_VEL
LIN {X 0,Y 121.939,Z 288.294,A -85,B 0,C 180,E1 -25518.526,E2 -25518.526} C_VEL
LIN {X 0,Y 121.971,Z 288.277,A -85,B 0,C 180,E1 -25524.821,E2 -25524.821} C_VEL
LIN {X 0,Y 121.924,Z 288.259,A -85,B 0,C 180,E1 -25529.84,E2 -25529.84} C_VEL
LIN {X 0,Y 121.979,Z 288.287,A -85,B 0,C 180,E1 -25536.219,E2 -25536.219} C_VEL
LIN {X 0,Y 122.04,Z 288.281,A -85,B 0,C 180,E1 -25539.79,E2 -25539.79} C_VEL
LIN {X 0,Y 122.218,Z 288.223,A -85,B 0,C 180,E1 -25546.706,E2 -25546.706} C_VEL
LIN {X 0,Y 122.398,Z 288.21,A -85,B 0,C 180,E1 -25550.085,E2 -25550.085} C_VEL
LIN {X 0,Y 122.596,Z 288.214,A -85,B 0,C 180,E1 -25556.718,E2 -25556.718} C_VEL
LIN {X 0,Y 123.04,Z 288.152,A -85,B 0,C 180,E1 -25560.004,E2 -25560.004} C_VEL
LIN {X 0,Y 122.442,Z 288.207,A -85,B 0,C 180,E1 -25566.596,E2 -25566.596} C_VEL
LIN {X 0,Y 122.445,Z 288.228,A -85,B 0,C 180,E1 -25569.919,E2 -25569.919} C_VEL
LIN {X 0,Y 122.265,Z 288.255,A -85,B 0,C 180,E1 -25573.297,E2 -25573.297} C_VEL
LIN {X 0,Y 122.051,Z 288.269,A -85,B 0,C 180,E1 -25580.216,E2 -25580.216} C_VEL
LIN {X 0,Y 121.986,Z 288.291,A -85,B 0,C 180,E1 -25583.788,E2 -25583.788} C_VEL
LIN {X 0,Y 121.93,Z 288.295,A -85,B 0,C 180,E1 -25590.164,E2 -25590.164} C_VEL
LIN {X 0,Y 121.901,Z 288.297,A -85,B 0,C 180,E1 -25596.182,E2 -25596.182} C_VEL
LIN {X 0,Y 122.112,Z 288.298,A -85,B 0,C 180,E1 -25601.047,E2 -25601.047} C_VEL
LIN {X 0,Y 122.406,Z 289.791,A -85,B 0,C 180,E1 -25603.996,E2 -25603.996} C_VEL
LIN {X 0,Y 123.454,Z 293,A -85,B 0,C 180,E1 -25604.671,E2 -25604.671} C_VEL
LIN {X 0,Y 126.844,Z 301.913,A -85,B 0,C 180,E1 -25606.811,E2 -25606.811} C_VEL
LIN {X 0,Y 128.539,Z 307.985,A -85,B 0,C 180,E1 -25608.221,E2 -25608.221} C_VEL
LIN {X 0,Y 129.754,Z 320.465,A -85,B 0,C 180,E1 -25611.009,E2 -25611.009} C_VEL
LIN {X 0,Y 130.445,Z 332.944,A -85,B 0,C 180,E1 -25614.324,E2 -25614.324} C_VEL
LIN {X 0,Y 130.379,Z 342.792,A -85,B 0,C 180,E1 -25617.382,E2 -25617.382} C_VEL
LIN {X 0,Y 130.116,Z 349.003,A -85,B 0,C 180,E1 -25619.579,E2 -25619.579} C_VEL
LIN {X 0,Y 126.721,Z 359.532,A -85,B 0,C 180,E1 -25623.661,E2 -25623.661} C_VEL
LIN {X 0,Y 124.269,Z 367.373,A -85,B 0,C 180,E1 -25627.558,E2 -25627.558} C_VEL
LIN {X 0,Y 121.855,Z 375.018,A -85,B 0,C 180,E1 -25632.374,E2 -25632.374} C_VEL
LIN {X 0,Y 120.223,Z 382.052,A -85,B 0,C 180,E1 -25638.193,E2 -25638.193} C_VEL
LIN {X 0,Y 119.559,Z 386.703,A -85,B 0,C 180,E1 -25643.248,E2 -25643.248} C_VEL
LIN {X 0,Y 119.429,Z 389.184,A -85,B 0,C 180,E1 -25646.626,E2 -25646.626} C_VEL
LIN {X 0,Y 119.494,Z 391.534,A -85,B 0,C 180,E1 -25650.757,E2 -25650.757} C_VEL
LIN {X 0,Y 119.448,Z 393.798,A -85,B 0,C 180,E1 -25656.757,E2 -25656.757} C_VEL
LIN {X 0,Y 120.606,Z 394.909,A -85,B 0,C 180,E1 -25663.478,E2 -25663.478} C_VEL
LIN {X 0,Y 123.226,Z 394.532,A -85,B 0,C 180,E1 -25670.01,E2 -25670.01} C_VEL
LIN {X 0,Y 127.64,Z 392.744,A -85,B 0,C 180,E1 -25676.134,E2 -25676.134} C_VEL
LIN {X 0,Y 130.375,Z 391.289,A -85,B 0,C 180,E1 -25679.021,E2 -25679.021} C_VEL
LIN {X 0,Y 136.675,Z 387.183,A -85,B 0,C 180,E1 -25684.445,E2 -25684.445} C_VEL
LIN {X 0,Y 142.203,Z 383.047,A -85,B 0,C 180,E1 -25688.153,E2 -25688.153} C_VEL
LIN {X 0,Y 148.392,Z 377.862,A -85,B 0,C 180,E1 -25691.532,E2 -25691.532} C_VEL
LIN {X 0,Y 154.034,Z 372.641,A -85,B 0,C 180,E1 -25694.089,E2 -25694.089} C_VEL
LIN {X 0,Y 156.393,Z 369.35,A -85,B 0,C 180,E1 -25695.971,E2 -25695.971} C_VEL
LIN {X 0,Y 159.119,Z 364.75,A -85,B 0,C 180,E1 -25698.663,E2 -25698.663} C_VEL
LIN {X 0,Y 160.137,Z 362.649,A -85,B 0,C 180,E1 -25699.984,E2 -25699.984} C_VEL
LIN {X 0,Y 160.767,Z 359.818,A -85,B 0,C 180,E1 -25702.261,E2 -25702.261} C_VEL
LIN {X 0,Y 161.223,Z 356.172,A -85,B 0,C 180,E1 -25705.916,E2 -25705.916} C_VEL
LIN {X 0,Y 161.356,Z 354.091,A -85,B 0,C 180,E1 -25708.485,E2 -25708.485} C_VEL
LIN {X 0,Y 161.348,Z 352.333,A -85,B 0,C 180,E1 -25711.368,E2 -25711.368} C_VEL
LIN {X 0,Y 161.678,Z 350.223,A -85,B 0,C 180,E1 -25715.899,E2 -25715.899} C_VEL
LIN {X 0,Y 161.999,Z 349.444,A -85,B 0,C 180,E1 -25719.689,E2 -25719.689} C_VEL
LIN {X 0,Y 161.789,Z 350.677,A -85,B 0,C 180,E1 -25724.889,E2 -25724.889} C_VEL
LIN {X 0,Y 162.112,Z 351.522,A -85,B 0,C 180,E1 -25727.478,E2 -25727.478} C_VEL
LIN {X 0,Y 162.162,Z 354.754,A -85,B 0,C 180,E1 -25732.526,E2 -25732.526} C_VEL
LIN {X 0,Y 161.525,Z 358.4,A -85,B 0,C 180,E1 -25736.255,E2 -25736.255} C_VEL
LIN {X 0,Y 160.505,Z 361.445,A -85,B 0,C 180,E1 -25738.743,E2 -25738.743} C_VEL
LIN {X 0,Y 159.691,Z 363.15,A -85,B 0,C 180,E1 -25739.964,E2 -25739.964} C_VEL
LIN {X 0,Y 158.407,Z 364.823,A -85,B 0,C 180,E1 -25740.822,E2 -25740.822} C_VEL
LIN {X 0,Y 155.303,Z 367.502,A -85,B 0,C 180,E1 -25741.596,E2 -25741.596} C_VEL
LIN {X 0,Y 147.543,Z 372.769,A -85,B 0,C 180,E1 -25742.701,E2 -25742.701} C_VEL
LIN {X 0,Y 144.67,Z 374.78,A -85,B 0,C 180,E1 -25743.594,E2 -25743.594} C_VEL
LIN {X 0,Y 137.729,Z 379.87,A -85,B 0,C 180,E1 -25747.263,E2 -25747.263} C_VEL
LIN {X 0,Y 132.268,Z 383.291,A -85,B 0,C 180,E1 -25750.714,E2 -25750.714} C_VEL
LIN {X 0,Y 125.345,Z 386.827,A -85,B 0,C 180,E1 -25756.277,E2 -25756.277} C_VEL
LIN {X 0,Y 120.652,Z 388.558,A -85,B 0,C 180,E1 -25761.255,E2 -25761.255} C_VEL
LIN {X 0,Y 117.298,Z 389.277,A -85,B 0,C 180,E1 -25766.011,E2 -25766.011} C_VEL
LIN {X 0,Y 114.772,Z 389.172,A -85,B 0,C 180,E1 -25770.99,E2 -25770.99} C_VEL
LIN {X 0,Y 112.977,Z 388.283,A -85,B 0,C 180,E1 -25776.034,E2 -25776.034} C_VEL
LIN {X 0,Y 111.946,Z 386.654,A -85,B 0,C 180,E1 -25781.12,E2 -25781.12} C_VEL
LIN {X 0,Y 111.665,Z 384.284,A -85,B 0,C 180,E1 -25786.188,E2 -25786.188} C_VEL
LIN {X 0,Y 112.196,Z 379.792,A -85,B 0,C 180,E1 -25792.854,E2 -25792.854} C_VEL
LIN {X 0,Y 113.324,Z 375.141,A -85,B 0,C 180,E1 -25798.011,E2 -25798.011} C_VEL
LIN {X 0,Y 115.248,Z 368.429,A -85,B 0,C 180,E1 -25803.762,E2 -25803.762} C_VEL
LIN {X 0,Y 117.828,Z 360.428,A -85,B 0,C 180,E1 -25809.031,E2 -25809.031} C_VEL
LIN {X 0,Y 121.104,Z 350.722,A -85,B 0,C 180,E1 -25813.913,E2 -25813.913} C_VEL
LIN {X 0,Y 124.308,Z 340.854,A -85,B 0,C 180,E1 -25817.76,E2 -25817.76} C_VEL
LIN {X 0,Y 125.671,Z 336.633,A -85,B 0,C 180,E1 -25819.121,E2 -25819.121} C_VEL
LIN {X 0,Y 125.096,Z 326,A -85,B 0,C 180,E1 -25822.739,E2 -25822.739} C_VEL
LIN {X 0,Y 124.041,Z 315.595,A -85,B 0,C 180,E1 -25825.842,E2 -25825.842} C_VEL
LIN {X 0,Y 122.331,Z 305.106,A -85,B 0,C 180,E1 -25828.672,E2 -25828.672} C_VEL
LIN {X 0,Y 118.441,Z 295.086,A -85,B 0,C 180,E1 -25831.647,E2 -25831.647} C_VEL
LIN {X 0,Y 116.926,Z 292.392,A -85,B 0,C 180,E1 -25832.542,E2 -25832.542} C_VEL
LIN {X 0,Y 115.634,Z 289.654,A -85,B 0,C 180,E1 -25833.365,E2 -25833.365} C_VEL
LIN {X 0,Y 115.551,Z 289.092,A -85,B 0,C 180,E1 -25833.487,E2 -25833.487} C_VEL
LIN {X 0,Y 115.363,Z 289.109,A -85,B 0,C 180,E1 -25840.531,E2 -25840.531} C_VEL
LIN {X 0,Y 115.155,Z 289.143,A -85,B 0,C 180,E1 -25844.13,E2 -25844.13} C_VEL
LIN {X 0,Y 114.995,Z 289.16,A -85,B 0,C 180,E1 -25851.512,E2 -25851.512} C_VEL
LIN {X 0,Y 114.867,Z 289.168,A -85,B 0,C 180,E1 -25855.359,E2 -25855.359} C_VEL
LIN {X 0,Y 114.856,Z 289.171,A -85,B 0,C 180,E1 -25861.066,E2 -25861.066} C_VEL
LIN {X 0,Y 114.881,Z 289.166,A -85,B 0,C 180,E1 -25867.717,E2 -25867.717} C_VEL
LIN {X 0,Y 114.874,Z 289.144,A -85,B 0,C 180,E1 -25872.77,E2 -25872.77} C_VEL
LIN {X 0,Y 114.866,Z 289.173,A -85,B 0,C 180,E1 -25877.705,E2 -25877.705} C_VEL
LIN {X 0,Y 114.851,Z 289.175,A -85,B 0,C 180,E1 -25882.702,E2 -25882.702} C_VEL
LIN {X 0,Y 114.859,Z 289.137,A -85,B 0,C 180,E1 -25888.94,E2 -25888.94} C_VEL
LIN {X 0,Y 114.944,Z 289.164,A -85,B 0,C 180,E1 -25896.511,E2 -25896.511} C_VEL
LIN {X 0,Y 115.005,Z 289.15,A -85,B 0,C 180,E1 -25902.213,E2 -25902.213} C_VEL
LIN {X 0,Y 115.232,Z 289.09,A -85,B 0,C 180,E1 -25907.376,E2 -25907.376} C_VEL
LIN {X 0,Y 115.362,Z 289.105,A -85,B 0,C 180,E1 -25913.006,E2 -25913.006} C_VEL
LIN {X 0,Y 115.992,Z 289.03,A -85,B 0,C 180,E1 -25920.004,E2 -25920.004} C_VEL
LIN {X 0,Y 115.385,Z 289.088,A -85,B 0,C 180,E1 -25927.001,E2 -25927.001} C_VEL
LIN {X 0,Y 115.285,Z 289.124,A -85,B 0,C 180,E1 -25932.74,E2 -25932.74} C_VEL
LIN {X 0,Y 115.019,Z 289.138,A -85,B 0,C 180,E1 -25937.793,E2 -25937.793} C_VEL
LIN {X 0,Y 114.95,Z 289.167,A -85,B 0,C 180,E1 -25943.497,E2 -25943.497} C_VEL
LIN {X 0,Y 114.86,Z 289.18,A -85,B 0,C 180,E1 -25951.061,E2 -25951.061} C_VEL
LIN {X 0,Y 114.853,Z 289.181,A -85,B 0,C 180,E1 -25957.733,E2 -25957.733} C_VEL
LIN {X 0,Y 115.076,Z 289.196,A -85,B 0,C 180,E1 -25961.041,E2 -25961.041} C_VEL
LIN {X 0,Y 115.158,Z 289.511,A -85,B 0,C 180,E1 -25961.734,E2 -25961.734} C_VEL
LIN {X 0,Y 116.24,Z 292.831,A -85,B 0,C 180,E1 -25962.495,E2 -25962.495} C_VEL
LIN {X 0,Y 119.688,Z 301.451,A -85,B 0,C 180,E1 -25964.805,E2 -25964.805} C_VEL
LIN {X 0,Y 122.128,Z 309.351,A -85,B 0,C 180,E1 -25966.905,E2 -25966.905} C_VEL
LIN {X 0,Y 123.154,Z 320.814,A -85,B 0,C 180,E1 -25969.677,E2 -25969.677} C_VEL
LIN {X 0,Y 123.659,Z 332.976,A -85,B 0,C 180,E1 -25973.102,E2 -25973.102} C_VEL
LIN {X 0,Y 123.573,Z 343.052,A -85,B 0,C 180,E1 -25976.421,E2 -25976.421} C_VEL
LIN {X 0,Y 123.367,Z 348.303,A -85,B 0,C 180,E1 -25978.382,E2 -25978.382} C_VEL
LIN {X 0,Y 120.91,Z 356.165,A -85,B 0,C 180,E1 -25981.454,E2 -25981.454} C_VEL
LIN {X 0,Y 117.706,Z 365.804,A -85,B 0,C 180,E1 -25986.232,E2 -25986.232} C_VEL
LIN {X 0,Y 115.117,Z 373.72,A -85,B 0,C 180,E1 -25991.306,E2 -25991.306} C_VEL
LIN {X 0,Y 113.688,Z 379.106,A -85,B 0,C 180,E1 -25995.684,E2 -25995.684} C_VEL
LIN {X 0,Y 112.693,Z 384.358,A -85,B 0,C 180,E1 -26001.03,E2 -26001.03} C_VEL
LIN {X 0,Y 112.352,Z 388.409,A -85,B 0,C 180,E1 -26006.413,E2 -26006.413} C_VEL
LIN {X 0,Y 112.455,Z 390.529,A -85,B 0,C 180,E1 -26009.999,E2 -26009.999} C_VEL
LIN {X 0,Y 112.339,Z 392.13,A -85,B 0,C 180,E1 -26013.586,E2 -26013.586} C_VEL
LIN {X 0,Y 112.858,Z 394.151,A -85,B 0,C 180,E1 -26020.766,E2 -26020.766} C_VEL
LIN {X 0,Y 114.934,Z 394.726,A -85,B 0,C 180,E1 -26027.802,E2 -26027.802} C_VEL
LIN {X 0,Y 118.728,Z 393.818,A -85,B 0,C 180,E1 -26034.478,E2 -26034.478} C_VEL
LIN {X 0,Y 124.198,Z 391.49,A -85,B 0,C 180,E1 -26040.615,E2 -26040.615} C_VEL
LIN {X 0,Y 129.125,Z 388.755,A -85,B 0,C 180,E1 -26044.853,E2 -26044.853} C_VEL
LIN {X 0,Y 136.732,Z 383.723,A -85,B 0,C 180,E1 -26049.977,E2 -26049.977} C_VEL
LIN {X 0,Y 143.208,Z 378.752,A -85,B 0,C 180,E1 -26053.396,E2 -26053.396} C_VEL
LIN {X 0,Y 149.024,Z 373.745,A -85,B 0,C 180,E1 -26055.986,E2 -26055.986} C_VEL
LIN {X 0,Y 152.316,Z 369.481,A -85,B 0,C 180,E1 -26058.688,E2 -26058.688} C_VEL
LIN {X 0,Y 154.295,Z 366.319,A -85,B 0,C 180,E1 -26060.743,E2 -26060.743} C_VEL
LIN {X 0,Y 155.17,Z 363.958,A -85,B 0,C 180,E1 -26062.758,E2 -26062.758} C_VEL
LIN {X 0,Y 155.782,Z 361.144,A -85,B 0,C 180,E1 -26065.796,E2 -26065.796} C_VEL
LIN {X 0,Y 156.135,Z 358.847,A -85,B 0,C 180,E1 -26068.783,E2 -26068.783} C_VEL
LIN {X 0,Y 156.436,Z 356.156,A -85,B 0,C 180,E1 -26073.961,E2 -26073.961} C_VEL
LIN {X 0,Y 156.762,Z 355.261,A -85,B 0,C 180,E1 -26076.2,E2 -26076.2} C_VEL
LIN {X 0,Y 157.046,Z 354.641,A -85,B 0,C 180,E1 -26080.009,E2 -26080.009} C_VEL
LIN {X 0,Y 156.989,Z 356.354,A -85,B 0,C 180,E1 -26087.063,E2 -26087.063} C_VEL
LIN {X 0,Y 156.751,Z 359.366,A -85,B 0,C 180,E1 -26092.267,E2 -26092.267} C_VEL
LIN {X 0,Y 156.119,Z 361.578,A -85,B 0,C 180,E1 -26094.831,E2 -26094.831} C_VEL
LIN {X 0,Y 155.027,Z 364.303,A -85,B 0,C 180,E1 -26097.399,E2 -26097.399} C_VEL
LIN {X 0,Y 153.646,Z 366.699,A -85,B 0,C 180,E1 -26099.276,E2 -26099.276} C_VEL
LIN {X 0,Y 152.82,Z 367.768,A -85,B 0,C 180,E1 -26099.997,E2 -26099.997} C_VEL
LIN {X 0,Y 144.67,Z 374.78,A -85,B 0,C 180,E1 -26103.594,E2 -26103.594} C_VEL
LIN {X 0,Y 140.863,Z 377.425,A -85,B 0,C 180,E1 -26105.091,E2 -26105.091} C_VEL
LIN {X 0,Y 130.348,Z 382.775,A -85,B 0,C 180,E1 -26108.201,E2 -26108.201} C_VEL
LIN {X 0,Y 124.739,Z 385.156,A -85,B 0,C 180,E1 -26110.444,E2 -26110.444} C_VEL
LIN {X 0,Y 122.501,Z 386.081,A -85,B 0,C 180,E1 -26111.859,E2 -26111.859} C_VEL
LIN {X 0,Y 116.17,Z 388.49,A -85,B 0,C 180,E1 -26117.603,E2 -26117.603} C_VEL
LIN {X 0,Y 112.527,Z 389.326,A -85,B 0,C 180,E1 -26122.003,E2 -26122.003} C_VEL
LIN {X 0,Y 109.517,Z 389.547,A -85,B 0,C 180,E1 -26126.688,E2 -26126.688} C_VEL
LIN {X 0,Y 107.271,Z 389.056,A -85,B 0,C 180,E1 -26131.604,E2 -26131.604} C_VEL
LIN {X 0,Y 105.568,Z 387.808,A -85,B 0,C 180,E1 -26136.98,E2 -26136.98} C_VEL
LIN {X 0,Y 104.714,Z 385.813,A -85,B 0,C 180,E1 -26142.417,E2 -26142.417} C_VEL
LIN {X 0,Y 104.602,Z 383.055,A -85,B 0,C 180,E1 -26147.789,E2 -26147.789} C_VEL
LIN {X 0,Y 105.177,Z 379.302,A -85,B 0,C 180,E1 -26153.298,E2 -26153.298} C_VEL
LIN {X 0,Y 106.447,Z 374.174,A -85,B 0,C 180,E1 -26159.117,E2 -26159.117} C_VEL
LIN {X 0,Y 108.541,Z 367.402,A -85,B 0,C 180,E1 -26165.014,E2 -26165.014} C_VEL
LIN {X 0,Y 111.154,Z 359.647,A -85,B 0,C 180,E1 -26170.222,E2 -26170.222} C_VEL
LIN {X 0,Y 114.259,Z 350.829,A -85,B 0,C 180,E1 -26174.847,E2 -26174.847} C_VEL
LIN {X 0,Y 117.535,Z 341.195,A -85,B 0,C 180,E1 -26178.795,E2 -26178.795} C_VEL
LIN {X 0,Y 118.926,Z 337.002,A -85,B 0,C 180,E1 -26180.219,E2 -26180.219} C_VEL
LIN {X 0,Y 118.415,Z 326.512,A -85,B 0,C 180,E1 -26184.039,E2 -26184.039} C_VEL
LIN {X 0,Y 117.568,Z 316.959,A -85,B 0,C 180,E1 -26187.112,E2 -26187.112} C_VEL
LIN {X 0,Y 116.458,Z 309.071,A -85,B 0,C 180,E1 -26189.407,E2 -26189.407} C_VEL
LIN {X 0,Y 113.415,Z 300.114,A -85,B 0,C 180,E1 -26192.266,E2 -26192.266} C_VEL
LIN {X 0,Y 109.733,Z 293.285,A -85,B 0,C 180,E1 -26194.794,E2 -26194.794} C_VEL
LIN {X 0,Y 108.504,Z 290.711,A -85,B 0,C 180,E1 -26195.692,E2 -26195.692} C_VEL
LIN {X 0,Y 108.373,Z 289.986,A -85,B 0,C 180,E1 -26196.05,E2 -26196.05} C_VEL
LIN {X 0,Y 108.208,Z 290.007,A -85,B 0,C 180,E1 -26203.056,E2 -26203.056} C_VEL
LIN {X 0,Y 107.917,Z 290.032,A -85,B 0,C 180,E1 -26209.003,E2 -26209.003} C_VEL
LIN {X 0,Y 107.86,Z 290.046,A -85,B 0,C 180,E1 -26214.199,E2 -26214.199} C_VEL
LIN {X 0,Y 107.789,Z 290.054,A -85,B 0,C 180,E1 -26222.056,E2 -26222.056} C_VEL
LIN {X 0,Y 107.782,Z 290.044,A -85,B 0,C 180,E1 -26228.521,E2 -26228.521} C_VEL
LIN {X 0,Y 107.768,Z 290.048,A -85,B 0,C 180,E1 -26235.836,E2 -26235.836} C_VEL
LIN {X 0,Y 107.751,Z 290.061,A -85,B 0,C 180,E1 -26241.507,E2 -26241.507} C_VEL
LIN {X 0,Y 107.801,Z 290.015,A -85,B 0,C 180,E1 -26248.569,E2 -26248.569} C_VEL
LIN {X 0,Y 107.908,Z 290.042,A -85,B 0,C 180,E1 -26257.002,E2 -26257.002} C_VEL
LIN {X 0,Y 108.021,Z 290.002,A -85,B 0,C 180,E1 -26264.92,E2 -26264.92} C_VEL
LIN {X 0,Y 108.219,Z 289.963,A -85,B 0,C 180,E1 -26268.77,E2 -26268.77} C_VEL
LIN {X 0,Y 108.299,Z 289.981,A -85,B 0,C 180,E1 -26272.547,E2 -26272.547} C_VEL
LIN {X 0,Y 108.942,Z 289.907,A -85,B 0,C 180,E1 -26280.004,E2 -26280.004} C_VEL
LIN {X 0,Y 108.326,Z 289.97,A -85,B 0,C 180,E1 -26287.46,E2 -26287.46} C_VEL
LIN {X 0,Y 108.2,Z 290.007,A -85,B 0,C 180,E1 -26293.019,E2 -26293.019} C_VEL
LIN {X 0,Y 107.91,Z 290.023,A -85,B 0,C 180,E1 -26299.009,E2 -26299.009} C_VEL
LIN {X 0,Y 107.86,Z 290.05,A -85,B 0,C 180,E1 -26304.187,E2 -26304.187} C_VEL
LIN {X 0,Y 107.785,Z 290.063,A -85,B 0,C 180,E1 -26312.043,E2 -26312.043} C_VEL
LIN {X 0,Y 107.882,Z 290.049,A -85,B 0,C 180,E1 -26319.2,E2 -26319.2} C_VEL
LIN {X 0,Y 108.929,Z 292.895,A -85,B 0,C 180,E1 -26320.032,E2 -26320.032} C_VEL
LIN {X 0,Y 109.941,Z 294.503,A -85,B 0,C 180,E1 -26320.64,E2 -26320.64} C_VEL
LIN {X 0,Y 113.74,Z 304.397,A -85,B 0,C 180,E1 -26323.59,E2 -26323.59} C_VEL
LIN {X 0,Y 115.934,Z 311.868,A -85,B 0,C 180,E1 -26325.75,E2 -26325.75} C_VEL
LIN {X 0,Y 116.668,Z 322.275,A -85,B 0,C 180,E1 -26328.499,E2 -26328.499} C_VEL
LIN {X 0,Y 116.979,Z 334.244,A -85,B 0,C 180,E1 -26332.168,E2 -26332.168} C_VEL
LIN {X 0,Y 116.75,Z 343.966,A -85,B 0,C 180,E1 -26335.643,E2 -26335.643} C_VEL
LIN {X 0,Y 116.396,Z 349.129,A -85,B 0,C 180,E1 -26337.713,E2 -26337.713} C_VEL
LIN {X 0,Y 112.862,Z 359.364,A -85,B 0,C 180,E1 -26342.158,E2 -26342.158} C_VEL
LIN {X 0,Y 110.197,Z 367.14,A -85,B 0,C 180,E1 -26346.509,E2 -26346.509} C_VEL
LIN {X 0,Y 107.66,Z 374.723,A -85,B 0,C 180,E1 -26351.936,E2 -26351.936} C_VEL
LIN {X 0,Y 105.968,Z 381.727,A -85,B 0,C 180,E1 -26358.523,E2 -26358.523} C_VEL
LIN {X 0,Y 105.355,Z 386.347,A -85,B 0,C 180,E1 -26364.257,E2 -26364.257} C_VEL
LIN {X 0,Y 105.389,Z 389.817,A -85,B 0,C 180,E1 -26369.999,E2 -26369.999} C_VEL
LIN {X 0,Y 105.287,Z 391.543,A -85,B 0,C 180,E1 -26373.827,E2 -26373.827} C_VEL
LIN {X 0,Y 105.893,Z 393.74,A -85,B 0,C 180,E1 -26381.484,E2 -26381.484} C_VEL
LIN {X 0,Y 108.159,Z 394.485,A -85,B 0,C 180,E1 -26388.958,E2 -26388.958} C_VEL
LIN {X 0,Y 112.291,Z 393.826,A -85,B 0,C 180,E1 -26395.982,E2 -26395.982} C_VEL
LIN {X 0,Y 118.133,Z 391.69,A -85,B 0,C 180,E1 -26402.372,E2 -26402.372} C_VEL
LIN {X 0,Y 125.235,Z 388.092,A -85,B 0,C 180,E1 -26408.118,E2 -26408.118} C_VEL
LIN {X 0,Y 131.391,Z 384.346,A -85,B 0,C 180,E1 -26411.959,E2 -26411.959} C_VEL
LIN {X 0,Y 138.186,Z 379.62,A -85,B 0,C 180,E1 -26415.398,E2 -26415.398} C_VEL
LIN {X 0,Y 143.043,Z 375.877,A -85,B 0,C 180,E1 -26417.473,E2 -26417.473} C_VEL
LIN {X 0,Y 145.029,Z 373.893,A -85,B 0,C 180,E1 -26418.686,E2 -26418.686} C_VEL
LIN {X 0,Y 148.041,Z 370.146,A -85,B 0,C 180,E1 -26421.311,E2 -26421.311} C_VEL
LIN {X 0,Y 148.787,Z 369.11,A -85,B 0,C 180,E1 -26422.113,E2 -26422.113} C_VEL
LIN {X 0,Y 149.654,Z 367.004,A -85,B 0,C 180,E1 -26424.247,E2 -26424.247} C_VEL
LIN {X 0,Y 150.361,Z 364.565,A -85,B 0,C 180,E1 -26427.279,E2 -26427.279} C_VEL
LIN {X 0,Y 150.677,Z 363.327,A -85,B 0,C 180,E1 -26429.128,E2 -26429.128} C_VEL
LIN {X 0,Y 151.366,Z 360.492,A -85,B 0,C 180,E1 -26435.296,E2 -26435.296} C_VEL
LIN {X 0,Y 151.702,Z 359.707,A -85,B 0,C 180,E1 -26438.243,E2 -26438.243} C_VEL
LIN {X 0,Y 151.763,Z 359.678,A -85,B 0,C 180,E1 -26441.082,E2 -26441.082} C_VEL
LIN {X 0,Y 151.63,Z 360.952,A -85,B 0,C 180,E1 -26446.735,E2 -26446.735} C_VEL
LIN {X 0,Y 151.387,Z 362.13,A -85,B 0,C 180,E1 -26449.295,E2 -26449.295} C_VEL
LIN {X 0,Y 151.098,Z 363.691,A -85,B 0,C 180,E1 -26451.976,E2 -26451.976} C_VEL
LIN {X 0,Y 150.23,Z 365.833,A -85,B 0,C 180,E1 -26454.628,E2 -26454.628} C_VEL
LIN {X 0,Y 148.642,Z 368.51,A -85,B 0,C 180,E1 -26457.287,E2 -26457.287} C_VEL
LIN {X 0,Y 147.284,Z 370.065,A -85,B 0,C 180,E1 -26458.401,E2 -26458.401} C_VEL
LIN {X 0,Y 139.009,Z 376.496,A -85,B 0,C 180,E1 -26461.947,E2 -26461.947} C_VEL
LIN {X 0,Y 130.943,Z 381.739,A -85,B 0,C 180,E1 -26466.159,E2 -26466.159} C_VEL
LIN {X 0,Y 125.441,Z 384.699,A -85,B 0,C 180,E1 -26469.672,E2 -26469.672} C_VEL
LIN {X 0,Y 122.501,Z 386.081,A -85,B 0,C 180,E1 -26471.859,E2 -26471.859} C_VEL
LIN {X 0,Y 119.09,Z 387.393,A -85,B 0,C 180,E1 -26474.067,E2 -26474.067} C_VEL
LIN {X 0,Y 112.307,Z 388.987,A -85,B 0,C 180,E1 -26477.574,E2 -26477.574} C_VEL
LIN {X 0,Y 105.966,Z 389.749,A -85,B 0,C 180,E1 -26481.561,E2 -26481.561} C_VEL
LIN {X 0,Y 103.372,Z 389.755,A -85,B 0,C 180,E1 -26484.468,E2 -26484.468} C_VEL
LIN {X 0,Y 99.774,Z 388.755,A -85,B 0,C 180,E1 -26492.302,E2 -26492.302} C_VEL
LIN {X 0,Y 97.833,Z 386.356,A -85,B 0,C 180,E1 -26500.274,E2 -26500.274} C_VEL
LIN {X 0,Y 97.536,Z 382.656,A -85,B 0,C 180,E1 -26507.897,E2 -26507.897} C_VEL
LIN {X 0,Y 98.379,Z 377.694,A -85,B 0,C 180,E1 -26515.146,E2 -26515.146} C_VEL
LIN {X 0,Y 100.021,Z 371.85,A -85,B 0,C 180,E1 -26521.564,E2 -26521.564} C_VEL
LIN {X 0,Y 102.49,Z 364.375,A -85,B 0,C 180,E1 -26527.844,E2 -26527.844} C_VEL
LIN {X 0,Y 105.854,Z 355.278,A -85,B 0,C 180,E1 -26533.611,E2 -26533.611} C_VEL
LIN {X 0,Y 109.489,Z 345.32,A -85,B 0,C 180,E1 -26538.429,E2 -26538.429} C_VEL
LIN {X 0,Y 112.115,Z 337.434,A -85,B 0,C 180,E1 -26541.439,E2 -26541.439} C_VEL
LIN {X 0,Y 111.789,Z 326.91,A -85,B 0,C 180,E1 -26545.493,E2 -26545.493} C_VEL
LIN {X 0,Y 110.836,Z 316.219,A -85,B 0,C 180,E1 -26549.13,E2 -26549.13} C_VEL
LIN {X 0,Y 109.995,Z 310.642,A -85,B 0,C 180,E1 -26550.917,E2 -26550.917} C_VEL
LIN {X 0,Y 107.27,Z 302.832,A -85,B 0,C 180,E1 -26553.757,E2 -26553.757} C_VEL
LIN {X 0,Y 102.583,Z 294.132,A -85,B 0,C 180,E1 -26557.38,E2 -26557.38} C_VEL
LIN {X 0,Y 101.34,Z 291.49,A -85,B 0,C 180,E1 -26558.412,E2 -26558.412} C_VEL
LIN {X 0,Y 101.242,Z 290.874,A -85,B 0,C 180,E1 -26558.735,E2 -26558.735} C_VEL
LIN {X 0,Y 101.13,Z 290.889,A -85,B 0,C 180,E1 -26563.386,E2 -26563.386} C_VEL
LIN {X 0,Y 100.825,Z 290.921,A -85,B 0,C 180,E1 -26570.397,E2 -26570.397} C_VEL
LIN {X 0,Y 100.767,Z 290.925,A -85,B 0,C 180,E1 -26574.961,E2 -26574.961} C_VEL
LIN {X 0,Y 100.702,Z 290.94,A -85,B 0,C 180,E1 -26583.135,E2 -26583.135} C_VEL
LIN {X 0,Y 100.721,Z 290.911,A -85,B 0,C 180,E1 -26589.874,E2 -26589.874} C_VEL
LIN {X 0,Y 100.735,Z 290.923,A -85,B 0,C 180,E1 -26595.766,E2 -26595.766} C_VEL
LIN {X 0,Y 100.692,Z 290.942,A -85,B 0,C 180,E1 -26601.091,E2 -26601.091} C_VEL
LIN {X 0,Y 100.701,Z 290.908,A -85,B 0,C 180,E1 -26606.876,E2 -26606.876} C_VEL
LIN {X 0,Y 100.782,Z 290.923,A -85,B 0,C 180,E1 -26615.271,E2 -26615.271} C_VEL
LIN {X 0,Y 100.812,Z 290.926,A -85,B 0,C 180,E1 -26619.605,E2 -26619.605} C_VEL
LIN {X 0,Y 101.087,Z 290.851,A -85,B 0,C 180,E1 -26626.739,E2 -26626.739} C_VEL
LIN {X 0,Y 101.233,Z 290.857,A -85,B 0,C 180,E1 -26632.024,E2 -26632.024} C_VEL
LIN {X 0,Y 101.865,Z 290.788,A -85,B 0,C 180,E1 -26640.005,E2 -26640.005} C_VEL
LIN {X 0,Y 101.265,Z 290.853,A -85,B 0,C 180,E1 -26647.983,E2 -26647.983} C_VEL
LIN {X 0,Y 101.126,Z 290.888,A -85,B 0,C 180,E1 -26653.355,E2 -26653.355} C_VEL
LIN {X 0,Y 100.821,Z 290.912,A -85,B 0,C 180,E1 -26660.403,E2 -26660.403} C_VEL
LIN {X 0,Y 100.778,Z 290.931,A -85,B 0,C 180,E1 -26664.963,E2 -26664.963} C_VEL
LIN {X 0,Y 100.699,Z 290.944,A -85,B 0,C 180,E1 -26673.123,E2 -26673.123} C_VEL
LIN {X 0,Y 100.71,Z 290.936,A -85,B 0,C 180,E1 -26676.388,E2 -26676.388} C_VEL
LIN {X 0,Y 101.875,Z 293.999,A -85,B 0,C 180,E1 -26677.447,E2 -26677.447} C_VEL
LIN {X 0,Y 103.222,Z 295.991,A -85,B 0,C 180,E1 -26678.315,E2 -26678.315} C_VEL
LIN {X 0,Y 105.071,Z 299.878,A -85,B 0,C 180,E1 -26679.773,E2 -26679.773} C_VEL
LIN {X 0,Y 108.355,Z 309.352,A -85,B 0,C 180,E1 -26682.93,E2 -26682.93} C_VEL
LIN {X 0,Y 109.532,Z 313.406,A -85,B 0,C 180,E1 -26684.255,E2 -26684.255} C_VEL
LIN {X 0,Y 110.155,Z 322.715,A -85,B 0,C 180,E1 -26686.936,E2 -26686.936} C_VEL
LIN {X 0,Y 110.325,Z 333.499,A -85,B 0,C 180,E1 -26690.43,E2 -26690.43} C_VEL
LIN {X 0,Y 110.1,Z 342.549,A -85,B 0,C 180,E1 -26693.811,E2 -26693.811} C_VEL
LIN {X 0,Y 109.504,Z 349.601,A -85,B 0,C 180,E1 -26696.805,E2 -26696.805} C_VEL
LIN {X 0,Y 105.973,Z 359.25,A -85,B 0,C 180,E1 -26701.262,E2 -26701.262} C_VEL
LIN {X 0,Y 103.175,Z 366.982,A -85,B 0,C 180,E1 -26705.876,E2 -26705.876} C_VEL
LIN {X 0,Y 100.575,Z 374.534,A -85,B 0,C 180,E1 -26711.672,E2 -26711.672} C_VEL
LIN {X 0,Y 99.014,Z 380.614,A -85,B 0,C 180,E1 -26717.705,E2 -26717.705} C_VEL
LIN {X 0,Y 98.301,Z 385.413,A -85,B 0,C 180,E1 -26723.843,E2 -26723.843} C_VEL
LIN {X 0,Y 98.313,Z 389.068,A -85,B 0,C 180,E1 -26729.999,E2 -26729.999} C_VEL
LIN {X 0,Y 98.232,Z 390.883,A -85,B 0,C 180,E1 -26734.102,E2 -26734.102} C_VEL
LIN {X 0,Y 98.93,Z 393.322,A -85,B 0,C 180,E1 -26742.304,E2 -26742.304} C_VEL
LIN {X 0,Y 101.437,Z 394.236,A -85,B 0,C 180,E1 -26750.268,E2 -26750.268} C_VEL
LIN {X 0,Y 105.945,Z 393.764,A -85,B 0,C 180,E1 -26757.667,E2 -26757.667} C_VEL
LIN {X 0,Y 112.194,Z 391.887,A -85,B 0,C 180,E1 -26764.316,E2 -26764.316} C_VEL
LIN {X 0,Y 119.739,Z 388.52,A -85,B 0,C 180,E1 -26770.212,E2 -26770.212} C_VEL
LIN {X 0,Y 126.231,Z 384.989,A -85,B 0,C 180,E1 -26774.101,E2 -26774.101} C_VEL
LIN {X 0,Y 133.346,Z 380.483,A -85,B 0,C 180,E1 -26777.549,E2 -26777.549} C_VEL
LIN {X 0,Y 138.332,Z 376.884,A -85,B 0,C 180,E1 -26779.646,E2 -26779.646} C_VEL
LIN {X 0,Y 140.326,Z 375.087,A -85,B 0,C 180,E1 -26780.92,E2 -26780.92} C_VEL
LIN {X 0,Y 142.031,Z 373.235,A -85,B 0,C 180,E1 -26782.344,E2 -26782.344} C_VEL
LIN {X 0,Y 143.451,Z 371.396,A -85,B 0,C 180,E1 -26783.988,E2 -26783.988} C_VEL
LIN {X 0,Y 144.623,Z 368.638,A -85,B 0,C 180,E1 -26787.683,E2 -26787.683} C_VEL
LIN {X 0,Y 145.136,Z 366.806,A -85,B 0,C 180,E1 -26791.034,E2 -26791.034} C_VEL
LIN {X 0,Y 145.963,Z 364.815,A -85,B 0,C 180,E1 -26796.179,E2 -26796.179} C_VEL
LIN {X 0,Y 146.137,Z 364.508,A -85,B 0,C 180,E1 -26797.369,E2 -26797.369} C_VEL
LIN {X 0,Y 146.301,Z 364.242,A -85,B 0,C 180,E1 -26800.347,E2 -26800.347} C_VEL
LIN {X 0,Y 146.023,Z 365.22,A -85,B 0,C 180,E1 -26806.072,E2 -26806.072} C_VEL
LIN {X 0,Y 145.743,Z 366.306,A -85,B 0,C 180,E1 -26808.875,E2 -26808.875} C_VEL
LIN {X 0,Y 145.231,Z 367.74,A -85,B 0,C 180,E1 -26811.649,E2 -26811.649} C_VEL
LIN {X 0,Y 144.08,Z 369.819,A -85,B 0,C 180,E1 -26814.398,E2 -26814.398} C_VEL
LIN {X 0,Y 142.427,Z 371.816,A -85,B 0,C 180,E1 -26816.442,E2 -26816.442} C_VEL
LIN {X 0,Y 133.529,Z 378.105,A -85,B 0,C 180,E1 -26820.127,E2 -26820.127} C_VEL
LIN {X 0,Y 124.232,Z 383.433,A -85,B 0,C 180,E1 -26824.919,E2 -26824.919} C_VEL
LIN {X 0,Y 115.995,Z 387.082,A -85,B 0,C 180,E1 -26830.468,E2 -26830.468} C_VEL
LIN {X 0,Y 109.731,Z 389.008,A -85,B 0,C 180,E1 -26836.119,E2 -26836.119} C_VEL
LIN {X 0,Y 105.527,Z 389.728,A -85,B 0,C 180,E1 -26841.194,E2 -26841.194} C_VEL
LIN {X 0,Y 103.372,Z 389.755,A -85,B 0,C 180,E1 -26844.468,E2 -26844.468} C_VEL
LIN {X 0,Y 101.04,Z 389.546,A -85,B 0,C 180,E1 -26847.503,E2 -26847.503} C_VEL
LIN {X 0,Y 96.061,Z 388.607,A -85,B 0,C 180,E1 -26852.456,E2 -26852.456} C_VEL
LIN {X 0,Y 92.442,Z 387.267,A -85,B 0,C 180,E1 -26856.705,E2 -26856.705} C_VEL
LIN {X 0,Y 90.805,Z 385.951,A -85,B 0,C 180,E1 -26860.183,E2 -26860.183} C_VEL
LIN {X 0,Y 90.586,Z 385.449,A -85,B 0,C 180,E1 -26861.39,E2 -26861.39} C_VEL
LIN {X 0,Y 90.466,Z 382.004,A -85,B 0,C 180,E1 -26868.399,E2 -26868.399} C_VEL
LIN {X 0,Y 91.459,Z 376.841,A -85,B 0,C 180,E1 -26876.148,E2 -26876.148} C_VEL
LIN {X 0,Y 93.309,Z 370.563,A -85,B 0,C 180,E1 -26883.134,E2 -26883.134} C_VEL
LIN {X 0,Y 96.1,Z 362.703,A -85,B 0,C 180,E1 -26889.789,E2 -26889.789} C_VEL
LIN {X 0,Y 99.589,Z 353.808,A -85,B 0,C 180,E1 -26895.507,E2 -26895.507} C_VEL
LIN {X 0,Y 103.209,Z 344.199,A -85,B 0,C 180,E1 -26900.199,E2 -26900.199} C_VEL
LIN {X 0,Y 105.158,Z 338.873,A -85,B 0,C 180,E1 -26902.319,E2 -26902.319} C_VEL
LIN {X 0,Y 105.309,Z 332.059,A -85,B 0,C 180,E1 -26905.215,E2 -26905.215} C_VEL
LIN {X 0,Y 104.854,Z 322.158,A -85,B 0,C 180,E1 -26909.04,E2 -26909.04} C_VEL
LIN {X 0,Y 103.962,Z 313.76,A -85,B 0,C 180,E1 -26912.03,E2 -26912.03} C_VEL
LIN {X 0,Y 101.434,Z 306.222,A -85,B 0,C 180,E1 -26915.069,E2 -26915.069} C_VEL
LIN {X 0,Y 95.755,Z 295.401,A -85,B 0,C 180,E1 -26920.121,E2 -26920.121} C_VEL
LIN {X 0,Y 94.408,Z 292.904,A -85,B 0,C 180,E1 -26921.337,E2 -26921.337} C_VEL
LIN {X 0,Y 94.155,Z 291.752,A -85,B 0,C 180,E1 -26921.846,E2 -26921.846} C_VEL
LIN {X 0,Y 93.796,Z 291.788,A -85,B 0,C 180,E1 -26927.441,E2 -26927.441} C_VEL
LIN {X 0,Y 93.696,Z 291.815,A -85,B 0,C 180,E1 -26932.027,E2 -26932.027} C_VEL
LIN {X 0,Y 93.614,Z 291.803,A -85,B 0,C 180,E1 -26936.772,E2 -26936.772} C_VEL
LIN {X 0,Y 93.616,Z 291.824,A -85,B 0,C 180,E1 -26944.341,E2 -26944.341} C_VEL
LIN {X 0,Y 93.638,Z 291.785,A -85,B 0,C 180,E1 -26952.492,E2 -26952.492} C_VEL
LIN {X 0,Y 93.625,Z 291.821,A -85,B 0,C 180,E1 -26958.646,E2 -26958.646} C_VEL
LIN {X 0,Y 93.608,Z 291.799,A -85,B 0,C 180,E1 -26965.676,E2 -26965.676} C_VEL
LIN {X 0,Y 93.665,Z 291.803,A -85,B 0,C 180,E1 -26974.21,E2 -26974.21} C_VEL
LIN {X 0,Y 93.689,Z 291.814,A -85,B 0,C 180,E1 -26977.977,E2 -26977.977} C_VEL
LIN {X 0,Y 94.007,Z 291.732,A -85,B 0,C 180,E1 -26986.379,E2 -26986.379} C_VEL
LIN {X 0,Y 94.163,Z 291.731,A -85,B 0,C 180,E1 -26991.42,E2 -26991.42} C_VEL
LIN {X 0,Y 94.791,Z 291.669,A -85,B 0,C 180,E1 -27000.005,E2 -27000.005} C_VEL
LIN {X 0,Y 94.199,Z 291.737,A -85,B 0,C 180,E1 -27008.587,E2 -27008.587} C_VEL
LIN {X 0,Y 94.044,Z 291.769,A -85,B 0,C 180,E1 -27013.712,E2 -27013.712} C_VEL
LIN {X 0,Y 93.698,Z 291.809,A -85,B 0,C 180,E1 -27022.032,E2 -27022.032} C_VEL
LIN {X 0,Y 93.623,Z 291.813,A -85,B 0,C 180,E1 -27026.775,E2 -27026.775} C_VEL
LIN {X 0,Y 93.657,Z 291.821,A -85,B 0,C 180,E1 -27033.25,E2 -27033.25} C_VEL
LIN {X 0,Y 94.639,Z 294.679,A -85,B 0,C 180,E1 -27034.306,E2 -27034.306} C_VEL
LIN {X 0,Y 95.968,Z 296.612,A -85,B 0,C 180,E1 -27035.316,E2 -27035.316} C_VEL
LIN {X 0,Y 99.398,Z 303.172,A -85,B 0,C 180,E1 -27038.225,E2 -27038.225} C_VEL
LIN {X 0,Y 102.383,Z 312.249,A -85,B 0,C 180,E1 -27041.577,E2 -27041.577} C_VEL
LIN {X 0,Y 103.512,Z 317.169,A -85,B 0,C 180,E1 -27043.334,E2 -27043.334} C_VEL
LIN {X 0,Y 103.744,Z 327.902,A -85,B 0,C 180,E1 -27046.793,E2 -27046.793} C_VEL
LIN {X 0,Y 103.534,Z 339.506,A -85,B 0,C 180,E1 -27051.178,E2 -27051.178} C_VEL
LIN {X 0,Y 102.811,Z 349.304,A -85,B 0,C 180,E1 -27055.498,E2 -27055.498} C_VEL
LIN {X 0,Y 99.131,Z 358.992,A -85,B 0,C 180,E1 -27060.246,E2 -27060.246} C_VEL
LIN {X 0,Y 96.181,Z 366.726,A -85,B 0,C 180,E1 -27065.155,E2 -27065.155} C_VEL
LIN {X 0,Y 93.493,Z 374.291,A -85,B 0,C 180,E1 -27071.368,E2 -27071.368} C_VEL
LIN {X 0,Y 91.714,Z 381.262,A -85,B 0,C 180,E1 -27078.955,E2 -27078.955} C_VEL
LIN {X 0,Y 91.182,Z 385.865,A -85,B 0,C 180,E1 -27085.579,E2 -27085.579} C_VEL
LIN {X 0,Y 91.247,Z 388.316,A -85,B 0,C 180,E1 -27089.999,E2 -27089.999} C_VEL
LIN {X 0,Y 91.175,Z 390.215,A -85,B 0,C 180,E1 -27094.42,E2 -27094.42} C_VEL
LIN {X 0,Y 92.002,Z 392.81,A -85,B 0,C 180,E1 -27103.247,E2 -27103.247} C_VEL
LIN {X 0,Y 94.778,Z 393.977,A -85,B 0,C 180,E1 -27111.762,E2 -27111.762} C_VEL
LIN {X 0,Y 99.705,Z 393.697,A -85,B 0,C 180,E1 -27119.564,E2 -27119.564} C_VEL
LIN {X 0,Y 106.403,Z 392.032,A -85,B 0,C 180,E1 -27126.472,E2 -27126.472} C_VEL
LIN {X 0,Y 114.411,Z 388.95,A -85,B 0,C 180,E1 -27132.507,E2 -27132.507} C_VEL
LIN {X 0,Y 121.269,Z 385.596,A -85,B 0,C 180,E1 -27136.419,E2 -27136.419} C_VEL
LIN {X 0,Y 128.707,Z 381.329,A -85,B 0,C 180,E1 -27139.857,E2 -27139.857} C_VEL
LIN {X 0,Y 133.82,Z 377.968,A -85,B 0,C 180,E1 -27141.976,E2 -27141.976} C_VEL
LIN {X 0,Y 135.782,Z 376.241,A -85,B 0,C 180,E1 -27143.346,E2 -27143.346} C_VEL
LIN {X 0,Y 137.412,Z 374.573,A -85,B 0,C 180,E1 -27144.915,E2 -27144.915} C_VEL
LIN {X 0,Y 138.561,Z 372.583,A -85,B 0,C 180,E1 -27147.819,E2 -27147.819} C_VEL
LIN {X 0,Y 138.964,Z 371.654,A -85,B 0,C 180,E1 -27149.616,E2 -27149.616} C_VEL
LIN {X 0,Y 139.926,Z 369.528,A -85,B 0,C 180,E1 -27154.696,E2 -27154.696} C_VEL
LIN {X 0,Y 140.247,Z 369.023,A -85,B 0,C 180,E1 -27156.363,E2 -27156.363} C_VEL
LIN {X 0,Y 140.53,Z 368.55,A -85,B 0,C 180,E1 -27159.505,E2 -27159.505} C_VEL
LIN {X 0,Y 140.387,Z 368.753,A -85,B 0,C 180,E1 -27162.517,E2 -27162.517} C_VEL
LIN {X 0,Y 140.243,Z 369.241,A -85,B 0,C 180,E1 -27165.486,E2 -27165.486} C_VEL
LIN {X 0,Y 139.912,Z 370.193,A -85,B 0,C 180,E1 -27168.406,E2 -27168.406} C_VEL
LIN {X 0,Y 139.205,Z 371.494,A -85,B 0,C 180,E1 -27171.285,E2 -27171.285} C_VEL
LIN {X 0,Y 137.627,Z 373.525,A -85,B 0,C 180,E1 -27174.135,E2 -27174.135} C_VEL
LIN {X 0,Y 136.076,Z 374.701,A -85,B 0,C 180,E1 -27174.959,E2 -27174.959} C_VEL
LIN {X 0,Y 126.524,Z 380.591,A -85,B 0,C 180,E1 -27178.888,E2 -27178.888} C_VEL
LIN {X 0,Y 117.763,Z 384.891,A -85,B 0,C 180,E1 -27183.417,E2 -27183.417} C_VEL
LIN {X 0,Y 111.879,Z 387.227,A -85,B 0,C 180,E1 -27187.213,E2 -27187.213} C_VEL
LIN {X 0,Y 106.558,Z 388.811,A -85,B 0,C 180,E1 -27191.407,E2 -27191.407} C_VEL
LIN {X 0,Y 101.952,Z 389.729,A -85,B 0,C 180,E1 -27196.001,E2 -27196.001} C_VEL
LIN {X 0,Y 96.66,Z 389.845,A -85,B 0,C 180,E1 -27203.163,E2 -27203.163} C_VEL
LIN {X 0,Y 94.647,Z 389.512,A -85,B 0,C 180,E1 -27206.997,E2 -27206.997} C_VEL
LIN {X 0,Y 92.281,Z 388.265,A -85,B 0,C 180,E1 -27213.1,E2 -27213.1} C_VEL
LIN {X 0,Y 90.586,Z 385.449,A -85,B 0,C 180,E1 -27221.39,E2 -27221.39} C_VEL
LIN {X 0,Y 89.712,Z 383.808,A -85,B 0,C 180,E1 -27224.949,E2 -27224.949} C_VEL
LIN {X 0,Y 88.192,Z 381.865,A -85,B 0,C 180,E1 -27228.432,E2 -27228.432} C_VEL
LIN {X 0,Y 85.088,Z 376.325,A -85,B 0,C 180,E1 -27236.669,E2 -27236.669} C_VEL
LIN {X 0,Y 85.246,Z 373.495,A -85,B 0,C 180,E1 -27240.224,E2 -27240.224} C_VEL
LIN {X 0,Y 87.715,Z 366.442,A -85,B 0,C 180,E1 -27247.511,E2 -27247.511} C_VEL
LIN {X 0,Y 90.451,Z 359.494,A -85,B 0,C 180,E1 -27253.061,E2 -27253.061} C_VEL
LIN {X 0,Y 94.041,Z 350.653,A -85,B 0,C 180,E1 -27258.537,E2 -27258.537} C_VEL
LIN {X 0,Y 98.068,Z 340.415,A -85,B 0,C 180,E1 -27263.315,E2 -27263.315} C_VEL
LIN {X 0,Y 98.567,Z 339.037,A -85,B 0,C 180,E1 -27263.863,E2 -27263.863} C_VEL
LIN {X 0,Y 98.657,Z 328.773,A -85,B 0,C 180,E1 -27268.47,E2 -27268.47} C_VEL
LIN {X 0,Y 98.066,Z 318.311,A -85,B 0,C 180,E1 -27272.643,E2 -27272.643} C_VEL
LIN {X 0,Y 96.4,Z 311.569,A -85,B 0,C 180,E1 -27275.494,E2 -27275.494} C_VEL
LIN {X 0,Y 91.198,Z 300.622,A -85,B 0,C 180,E1 -27281.106,E2 -27281.106} C_VEL
LIN {X 0,Y 88.178,Z 295.812,A -85,B 0,C 180,E1 -27284.019,E2 -27284.019} C_VEL
LIN {X 0,Y 86.931,Z 293.151,A -85,B 0,C 180,E1 -27285.42,E2 -27285.42} C_VEL
LIN {X 0,Y 86.841,Z 292.662,A -85,B 0,C 180,E1 -27285.639,E2 -27285.639} C_VEL
LIN {X 0,Y 86.584,Z 292.697,A -85,B 0,C 180,E1 -27293.944,E2 -27293.944} C_VEL
LIN {X 0,Y 86.472,Z 292.691,A -85,B 0,C 180,E1 -27299.186,E2 -27299.186} C_VEL
LIN {X 0,Y 86.545,Z 292.703,A -85,B 0,C 180,E1 -27305.712,E2 -27305.712} C_VEL
LIN {X 0,Y 86.563,Z 292.666,A -85,B 0,C 180,E1 -27313.063,E2 -27313.063} C_VEL
LIN {X 0,Y 86.549,Z 292.704,A -85,B 0,C 180,E1 -27319.495,E2 -27319.495} C_VEL
LIN {X 0,Y 86.556,Z 292.679,A -85,B 0,C 180,E1 -27325.37,E2 -27325.37} C_VEL
LIN {X 0,Y 86.58,Z 292.678,A -85,B 0,C 180,E1 -27333.24,E2 -27333.24} C_VEL
LIN {X 0,Y 86.641,Z 292.687,A -85,B 0,C 180,E1 -27341.073,E2 -27341.073} C_VEL
LIN {X 0,Y 86.929,Z 292.615,A -85,B 0,C 180,E1 -27345.969,E2 -27345.969} C_VEL
LIN {X 0,Y 87.056,Z 292.607,A -85,B 0,C 180,E1 -27350.714,E2 -27350.714} C_VEL
LIN {X 0,Y 87.717,Z 292.55,A -85,B 0,C 180,E1 -27360.005,E2 -27360.005} C_VEL
LIN {X 0,Y 87.107,Z 292.624,A -85,B 0,C 180,E1 -27369.292,E2 -27369.292} C_VEL
LIN {X 0,Y 86.952,Z 292.651,A -85,B 0,C 180,E1 -27374.093,E2 -27374.093} C_VEL
LIN {X 0,Y 86.59,Z 292.7,A -85,B 0,C 180,E1 -27383.948,E2 -27383.948} C_VEL
LIN {X 0,Y 86.493,Z 292.701,A -85,B 0,C 180,E1 -27389.351,E2 -27389.351} C_VEL
LIN {X 0,Y 87.53,Z 295.59,A -85,B 0,C 180,E1 -27390.627,E2 -27390.627} C_VEL
LIN {X 0,Y 89.099,Z 297.664,A -85,B 0,C 180,E1 -27392.009,E2 -27392.009} C_VEL
LIN {X 0,Y 93.908,Z 306.946,A -85,B 0,C 180,E1 -27396.784,E2 -27396.784} C_VEL
LIN {X 0,Y 96.799,Z 316.69,A -85,B 0,C 180,E1 -27400.807,E2 -27400.807} C_VEL
LIN {X 0,Y 97.335,Z 320.743,A -85,B 0,C 180,E1 -27402.307,E2 -27402.307} C_VEL
LIN {X 0,Y 97.193,Z 331.856,A -85,B 0,C 180,E1 -27406.317,E2 -27406.317} C_VEL
LIN {X 0,Y 96.671,Z 343.03,A -85,B 0,C 180,E1 -27411.095,E2 -27411.095} C_VEL
LIN {X 0,Y 96.038,Z 349.323,A -85,B 0,C 180,E1 -27414.166,E2 -27414.166} C_VEL
LIN {X 0,Y 92.311,Z 358.729,A -85,B 0,C 180,E1 -27419.076,E2 -27419.076} C_VEL
LIN {X 0,Y 89.2,Z 366.469,A -85,B 0,C 180,E1 -27424.32,E2 -27424.32} C_VEL
LIN {X 0,Y 86.412,Z 374.047,A -85,B 0,C 180,E1 -27431.014,E2 -27431.014} C_VEL
LIN {X 0,Y 84.752,Z 380.113,A -85,B 0,C 180,E1 -27438.035,E2 -27438.035} C_VEL
LIN {X 0,Y 84.13,Z 384.899,A -85,B 0,C 180,E1 -27445.207,E2 -27445.207} C_VEL
LIN {X 0,Y 84.182,Z 387.446,A -85,B 0,C 180,E1 -27449.999,E2 -27449.999} C_VEL
LIN {X 0,Y 84.138,Z 389.491,A -85,B 0,C 180,E1 -27454.791,E2 -27454.791} C_VEL
LIN {X 0,Y 85.111,Z 392.292,A -85,B 0,C 180,E1 -27464.342,E2 -27464.342} C_VEL
LIN {X 0,Y 88.198,Z 393.638,A -85,B 0,C 180,E1 -27473.478,E2 -27473.478} C_VEL
LIN {X 0,Y 93.591,Z 393.62,A -85,B 0,C 180,E1 -27481.711,E2 -27481.711} C_VEL
LIN {X 0,Y 100.782,Z 392.167,A -85,B 0,C 180,E1 -27488.873,E2 -27488.873} C_VEL
LIN {X 0,Y 109.29,Z 389.31,A -85,B 0,C 180,E1 -27495.019,E2 -27495.019} C_VEL
LIN {X 0,Y 116.506,Z 386.191,A -85,B 0,C 180,E1 -27498.94,E2 -27498.94} C_VEL
LIN {X 0,Y 127.021,Z 380.596,A -85,B 0,C 180,E1 -27503.346,E2 -27503.346} C_VEL
LIN {X 0,Y 129.452,Z 378.958,A -85,B 0,C 180,E1 -27504.521,E2 -27504.521} C_VEL
LIN {X 0,Y 131.251,Z 377.528,A -85,B 0,C 180,E1 -27505.93,E2 -27505.93} C_VEL
LIN {X 0,Y 132.359,Z 376.102,A -85,B 0,C 180,E1 -27508.162,E2 -27508.162} C_VEL
LIN {X 0,Y 133.606,Z 373.902,A -85,B 0,C 180,E1 -27513.408,E2 -27513.408} C_VEL
LIN {X 0,Y 134.042,Z 373.298,A -85,B 0,C 180,E1 -27515.196,E2 -27515.196} C_VEL
LIN {X 0,Y 134.479,Z 372.622,A -85,B 0,C 180,E1 -27518.538,E2 -27518.538} C_VEL
LIN {X 0,Y 134.533,Z 372.582,A -85,B 0,C 180,E1 -27521.73,E2 -27521.73} C_VEL
LIN {X 0,Y 134.28,Z 372.996,A -85,B 0,C 180,E1 -27524.826,E2 -27524.826} C_VEL
LIN {X 0,Y 133.894,Z 373.769,A -85,B 0,C 180,E1 -27527.877,E2 -27527.877} C_VEL
LIN {X 0,Y 132.999,Z 374.992,A -85,B 0,C 180,E1 -27530.875,E2 -27530.875} C_VEL
LIN {X 0,Y 132.12,Z 375.896,A -85,B 0,C 180,E1 -27532.354,E2 -27532.354} C_VEL
LIN {X 0,Y 127.123,Z 378.91,A -85,B 0,C 180,E1 -27534.329,E2 -27534.329} C_VEL
LIN {X 0,Y 117.216,Z 383.886,A -85,B 0,C 180,E1 -27538.606,E2 -27538.606} C_VEL
LIN {X 0,Y 108.15,Z 387.381,A -85,B 0,C 180,E1 -27543.721,E2 -27543.721} C_VEL
LIN {X 0,Y 99.891,Z 389.497,A -85,B 0,C 180,E1 -27549.949,E2 -27549.949} C_VEL
LIN {X 0,Y 92.731,Z 390.232,A -85,B 0,C 180,E1 -27557.642,E2 -27557.642} C_VEL
LIN {X 0,Y 89.103,Z 389.855,A -85,B 0,C 180,E1 -27563.221,E2 -27563.221} C_VEL
LIN {X 0,Y 86.341,Z 388.852,A -85,B 0,C 180,E1 -27569.228,E2 -27569.228} C_VEL
LIN {X 0,Y 84.393,Z 387.077,A -85,B 0,C 180,E1 -27575.65,E2 -27575.65} C_VEL
LIN {X 0,Y 83.317,Z 383.355,A -85,B 0,C 180,E1 -27584.987,E2 -27584.987} C_VEL
LIN {X 0,Y 83.638,Z 379.66,A -85,B 0,C 180,E1 -27591.736,E2 -27591.736} C_VEL
LIN {X 0,Y 84.815,Z 374.981,A -85,B 0,C 180,E1 -27598.41,E2 -27598.41} C_VEL
LIN {X 0,Y 85.246,Z 373.495,A -85,B 0,C 180,E1 -27600.224,E2 -27600.224} C_VEL
LIN {X 0,Y 85.561,Z 370.502,A -85,B 0,C 180,E1 -27603.636,E2 -27603.636} C_VEL
LIN {X 0,Y 84.692,Z 365.017,A -85,B 0,C 180,E1 -27609.184,E2 -27609.184} C_VEL
LIN {X 0,Y 84.367,Z 358.899,A -85,B 0,C 180,E1 -27614.526,E2 -27614.526} C_VEL
LIN {X 0,Y 85.494,Z 354.906,A -85,B 0,C 180,E1 -27617.397,E2 -27617.397} C_VEL
LIN {X 0,Y 89.494,Z 345.634,A -85,B 0,C 180,E1 -27622.671,E2 -27622.671} C_VEL
LIN {X 0,Y 91.969,Z 339.165,A -85,B 0,C 180,E1 -27625.618,E2 -27625.618} C_VEL
LIN {X 0,Y 92.159,Z 328.91,A -85,B 0,C 180,E1 -27630.547,E2 -27630.547} C_VEL
LIN {X 0,Y 91.673,Z 319.192,A -85,B 0,C 180,E1 -27634.778,E2 -27634.778} C_VEL
LIN {X 0,Y 90.291,Z 314.267,A -85,B 0,C 180,E1 -27637.226,E2 -27637.226} C_VEL
LIN {X 0,Y 86.293,Z 305.554,A -85,B 0,C 180,E1 -27642.255,E2 -27642.255} C_VEL
LIN {X 0,Y 82.096,Z 298.039,A -85,B 0,C 180,E1 -27647.221,E2 -27647.221} C_VEL
LIN {X 0,Y 80.086,Z 295.454,A -85,B 0,C 180,E1 -27649.425,E2 -27649.425} C_VEL
LIN {X 0,Y 79.538,Z 293.572,A -85,B 0,C 180,E1 -27650.512,E2 -27650.512} C_VEL
LIN {X 0,Y 79.476,Z 293.56,A -85,B 0,C 180,E1 -27657.849,E2 -27657.849} C_VEL
LIN {X 0,Y 79.456,Z 293.578,A -85,B 0,C 180,E1 -27667.255,E2 -27667.255} C_VEL
LIN {X 0,Y 79.466,Z 293.561,A -85,B 0,C 180,E1 -27675.033,E2 -27675.033} C_VEL
LIN {X 0,Y 79.448,Z 293.582,A -85,B 0,C 180,E1 -27682.763,E2 -27682.763} C_VEL
LIN {X 0,Y 79.478,Z 293.55,A -85,B 0,C 180,E1 -27692.161,E2 -27692.161} C_VEL
LIN {X 0,Y 79.509,Z 293.58,A -85,B 0,C 180,E1 -27699.301,E2 -27699.301} C_VEL
LIN {X 0,Y 79.821,Z 293.501,A -85,B 0,C 180,E1 -27705.582,E2 -27705.582} C_VEL
LIN {X 0,Y 79.946,Z 293.484,A -85,B 0,C 180,E1 -27709.88,E2 -27709.88} C_VEL
LIN {X 0,Y 80.644,Z 293.431,A -85,B 0,C 180,E1 -27720.006,E2 -27720.006} C_VEL
LIN {X 0,Y 79.993,Z 293.515,A -85,B 0,C 180,E1 -27730.126,E2 -27730.126} C_VEL
LIN {X 0,Y 79.765,Z 293.539,A -85,B 0,C 180,E1 -27735.333,E2 -27735.333} C_VEL
LIN {X 0,Y 79.548,Z 293.759,A -85,B 0,C 180,E1 -27744.819,E2 -27744.819} C_VEL
LIN {X 0,Y 80.556,Z 296.408,A -85,B 0,C 180,E1 -27746.281,E2 -27746.281} C_VEL
LIN {X 0,Y 82.086,Z 298.649,A -85,B 0,C 180,E1 -27747.999,E2 -27747.999} C_VEL
LIN {X 0,Y 86.67,Z 307.085,A -85,B 0,C 180,E1 -27753.192,E2 -27753.192} C_VEL
LIN {X 0,Y 88.73,Z 311.742,A -85,B 0,C 180,E1 -27755.749,E2 -27755.749} C_VEL
LIN {X 0,Y 91.033,Z 320.992,A -85,B 0,C 180,E1 -27759.997,E2 -27759.997} C_VEL
LIN {X 0,Y 90.745,Z 332.473,A -85,B 0,C 180,E1 -27764.495,E2 -27764.495} C_VEL
LIN {X 0,Y 89.946,Z 344.026,A -85,B 0,C 180,E1 -27769.863,E2 -27769.863} C_VEL
LIN {X 0,Y 89.169,Z 349.939,A -85,B 0,C 180,E1 -27772.971,E2 -27772.971} C_VEL
LIN {X 0,Y 85.557,Z 358.404,A -85,B 0,C 180,E1 -27777.728,E2 -27777.728} C_VEL
LIN {X 0,Y 82.258,Z 366.129,A -85,B 0,C 180,E1 -27783.349,E2 -27783.349} C_VEL
LIN {X 0,Y 79.335,Z 373.712,A -85,B 0,C 180,E1 -27790.597,E2 -27790.597} C_VEL
LIN {X 0,Y 77.461,Z 380.673,A -85,B 0,C 180,E1 -27799.545,E2 -27799.545} C_VEL
LIN {X 0,Y 77.075,Z 385.28,A -85,B 0,C 180,E1 -27807.386,E2 -27807.386} C_VEL
LIN {X 0,Y 77.09,Z 387.707,A -85,B 0,C 180,E1 -27812.612,E2 -27812.612} C_VEL
LIN {X 0,Y 77.344,Z 390.408,A -85,B 0,C 180,E1 -27820.47,E2 -27820.47} C_VEL
LIN {X 0,Y 79.708,Z 392.697,A -85,B 0,C 180,E1 -27830.65,E2 -27830.65} C_VEL
LIN {X 0,Y 84.397,Z 393.548,A -85,B 0,C 180,E1 -27839.975,E2 -27839.975} C_VEL
LIN {X 0,Y 91.257,Z 393.043,A -85,B 0,C 180,E1 -27848.031,E2 -27848.031} C_VEL
LIN {X 0,Y 99.742,Z 391.172,A -85,B 0,C 180,E1 -27854.797,E2 -27854.797} C_VEL
LIN {X 0,Y 109.382,Z 387.826,A -85,B 0,C 180,E1 -27860.444,E2 -27860.444} C_VEL
LIN {X 0,Y 120.128,Z 382.959,A -85,B 0,C 180,E1 -27864.989,E2 -27864.989} C_VEL
LIN {X 0,Y 122.926,Z 381.468,A -85,B 0,C 180,E1 -27865.994,E2 -27865.994} C_VEL
LIN {X 0,Y 125.253,Z 380.039,A -85,B 0,C 180,E1 -27867.313,E2 -27867.313} C_VEL
LIN {X 0,Y 126.372,Z 378.713,A -85,B 0,C 180,E1 -27869.961,E2 -27869.961} C_VEL
LIN {X 0,Y 127.452,Z 377.332,A -85,B 0,C 180,E1 -27873.82,E2 -27873.82} C_VEL
LIN {X 0,Y 128.347,Z 376.255,A -85,B 0,C 180,E1 -27878.568,E2 -27878.568} C_VEL
LIN {X 0,Y 128.448,Z 376.155,A -85,B 0,C 180,E1 -27880.831,E2 -27880.831} C_VEL
LIN {X 0,Y 128.167,Z 376.454,A -85,B 0,C 180,E1 -27884.083,E2 -27884.083} C_VEL
LIN {X 0,Y 127.712,Z 377.05,A -85,B 0,C 180,E1 -27887.28,E2 -27887.28} C_VEL
LIN {X 0,Y 126.603,Z 378.203,A -85,B 0,C 180,E1 -27890.41,E2 -27890.41} C_VEL
LIN {X 0,Y 115.87,Z 383.478,A -85,B 0,C 180,E1 -27894.525,E2 -27894.525} C_VEL
LIN {X 0,Y 105.419,Z 387.372,A -85,B 0,C 180,E1 -27899.671,E2 -27899.671} C_VEL
LIN {X 0,Y 98.511,Z 389.175,A -85,B 0,C 180,E1 -27904.086,E2 -27904.086} C_VEL
LIN {X 0,Y 92.5,Z 390.179,A -85,B 0,C 180,E1 -27908.999,E2 -27908.999} C_VEL
LIN {X 0,Y 87.165,Z 390.467,A -85,B 0,C 180,E1 -27914.644,E2 -27914.644} C_VEL
LIN {X 0,Y 82.787,Z 389.952,A -85,B 0,C 180,E1 -27920.967,E2 -27920.967} C_VEL
LIN {X 0,Y 79.512,Z 388.686,A -85,B 0,C 180,E1 -27927.888,E2 -27927.888} C_VEL
LIN {X 0,Y 77.327,Z 386.691,A -85,B 0,C 180,E1 -27935.12,E2 -27935.12} C_VEL
LIN {X 0,Y 76.253,Z 382.7,A -85,B 0,C 180,E1 -27945.245,E2 -27945.245} C_VEL
LIN {X 0,Y 77.008,Z 377.177,A -85,B 0,C 180,E1 -27955.211,E2 -27955.211} C_VEL
LIN {X 0,Y 79.002,Z 370.821,A -85,B 0,C 180,E1 -27963.591,E2 -27963.591} C_VEL
LIN {X 0,Y 81.821,Z 363.55,A -85,B 0,C 180,E1 -27970.862,E2 -27970.862} C_VEL
LIN {X 0,Y 85.494,Z 354.906,A -85,B 0,C 180,E1 -27977.397,E2 -27977.397} C_VEL
LIN {X 0,Y 86.26,Z 352.167,A -85,B 0,C 180,E1 -27979.21,E2 -27979.21} C_VEL
LIN {X 0,Y 86.134,Z 347.525,A -85,B 0,C 180,E1 -27982.365,E2 -27982.365} C_VEL
LIN {X 0,Y 85.377,Z 339.674,A -85,B 0,C 180,E1 -27987.394,E2 -27987.394} C_VEL
LIN {X 0,Y 85.76,Z 329.051,A -85,B 0,C 180,E1 -27992.937,E2 -27992.937} C_VEL
LIN {X 0,Y 85.511,Z 321.646,A -85,B 0,C 180,E1 -27996.497,E2 -27996.497} C_VEL
LIN {X 0,Y 84.266,Z 317.238,A -85,B 0,C 180,E1 -27999.003,E2 -27999.003} C_VEL
LIN {X 0,Y 80.019,Z 307.726,A -85,B 0,C 180,E1 -28005.278,E2 -28005.278} C_VEL
LIN {X 0,Y 77.744,Z 303.441,A -85,B 0,C 180,E1 -28008.531,E2 -28008.531} C_VEL
LIN {X 0,Y 75.539,Z 300.101,A -85,B 0,C 180,E1 -28011.525,E2 -28011.525} C_VEL
LIN {X 0,Y 75.341,Z 299.517,A -85,B 0,C 180,E1 -28011.909,E2 -28011.909} C_VEL
LIN {X 0,Y 73.165,Z 296.871,A -85,B 0,C 180,E1 -28014.833,E2 -28014.833} C_VEL
LIN {X 0,Y 72.468,Z 294.435,A -85,B 0,C 180,E1 -28016.456,E2 -28016.456} C_VEL
LIN {X 0,Y 72.339,Z 294.472,A -85,B 0,C 180,E1 -28025.657,E2 -28025.657} C_VEL
LIN {X 0,Y 72.312,Z 294.438,A -85,B 0,C 180,E1 -28032.869,E2 -28032.869} C_VEL
LIN {X 0,Y 72.355,Z 294.472,A -85,B 0,C 180,E1 -28040.992,E2 -28040.992} C_VEL
LIN {X 0,Y 72.333,Z 294.455,A -85,B 0,C 180,E1 -28044.349,E2 -28044.349} C_VEL
LIN {X 0,Y 72.388,Z 294.423,A -85,B 0,C 180,E1 -28050.967,E2 -28050.967} C_VEL
LIN {X 0,Y 72.39,Z 294.466,A -85,B 0,C 180,E1 -28057.156,E2 -28057.156} C_VEL
LIN {X 0,Y 72.719,Z 294.386,A -85,B 0,C 180,E1 -28065.119,E2 -28065.119} C_VEL
LIN {X 0,Y 72.843,Z 294.363,A -85,B 0,C 180,E1 -28068.881,E2 -28068.881} C_VEL
LIN {X 0,Y 73.569,Z 294.31,A -85,B 0,C 180,E1 -28080.007,E2 -28080.007} C_VEL
LIN {X 0,Y 72.881,Z 294.405,A -85,B 0,C 180,E1 -28091.127,E2 -28091.127} C_VEL
LIN {X 0,Y 72.585,Z 294.421,A -85,B 0,C 180,E1 -28096.893,E2 -28096.893} C_VEL
LIN {X 0,Y 72.49,Z 294.453,A -85,B 0,C 180,E1 -28098.739,E2 -28098.739} C_VEL
LIN {X 0,Y 73.279,Z 296.932,A -85,B 0,C 180,E1 -28100.351,E2 -28100.351} C_VEL
LIN {X 0,Y 75.395,Z 299.675,A -85,B 0,C 180,E1 -28103.164,E2 -28103.164} C_VEL
LIN {X 0,Y 80.569,Z 309.518,A -85,B 0,C 180,E1 -28110.486,E2 -28110.486} C_VEL
LIN {X 0,Y 82.931,Z 314.742,A -85,B 0,C 180,E1 -28113.796,E2 -28113.796} C_VEL
LIN {X 0,Y 84.722,Z 322.253,A -85,B 0,C 180,E1 -28117.666,E2 -28117.666} C_VEL
LIN {X 0,Y 84.846,Z 325.928,A -85,B 0,C 180,E1 -28119.315,E2 -28119.315} C_VEL
LIN {X 0,Y 83.968,Z 337.745,A -85,B 0,C 180,E1 -28124.648,E2 -28124.648} C_VEL
LIN {X 0,Y 83.121,Z 345.913,A -85,B 0,C 180,E1 -28128.977,E2 -28128.977} C_VEL
LIN {X 0,Y 82.593,Z 349.446,A -85,B 0,C 180,E1 -28131.031,E2 -28131.031} C_VEL
LIN {X 0,Y 78.84,Z 357.986,A -85,B 0,C 180,E1 -28136.142,E2 -28136.142} C_VEL
LIN {X 0,Y 75.353,Z 365.748,A -85,B 0,C 180,E1 -28142.203,E2 -28142.203} C_VEL
LIN {X 0,Y 72.267,Z 373.369,A -85,B 0,C 180,E1 -28150.1,E2 -28150.1} C_VEL
LIN {X 0,Y 70.496,Z 379.465,A -85,B 0,C 180,E1 -28158.498,E2 -28158.498} C_VEL
LIN {X 0,Y 70.021,Z 384.282,A -85,B 0,C 180,E1 -28167.123,E2 -28167.123} C_VEL
LIN {X 0,Y 70.067,Z 386.798,A -85,B 0,C 180,E1 -28172.874,E2 -28172.874} C_VEL
LIN {X 0,Y 70.401,Z 389.67,A -85,B 0,C 180,E1 -28181.516,E2 -28181.516} C_VEL
LIN {X 0,Y 73.087,Z 392.176,A -85,B 0,C 180,E1 -28192.62,E2 -28192.62} C_VEL
LIN {X 0,Y 78.329,Z 393.29,A -85,B 0,C 180,E1 -28202.569,E2 -28202.569} C_VEL
LIN {X 0,Y 85.768,Z 392.996,A -85,B 0,C 180,E1 -28210.959,E2 -28210.959} C_VEL
LIN {X 0,Y 94.822,Z 391.344,A -85,B 0,C 180,E1 -28217.83,E2 -28217.83} C_VEL
LIN {X 0,Y 105.018,Z 388.321,A -85,B 0,C 180,E1 -28223.421,E2 -28223.421} C_VEL
LIN {X 0,Y 116.236,Z 383.73,A -85,B 0,C 180,E1 -28227.829,E2 -28227.829} C_VEL
LIN {X 0,Y 119.031,Z 382.383,A -85,B 0,C 180,E1 -28228.882,E2 -28228.882} C_VEL
LIN {X 0,Y 120.474,Z 381.026,A -85,B 0,C 180,E1 -28232.176,E2 -28232.176} C_VEL
LIN {X 0,Y 121.775,Z 379.745,A -85,B 0,C 180,E1 -28237.425,E2 -28237.425} C_VEL
LIN {X 0,Y 122.09,Z 379.463,A -85,B 0,C 180,E1 -28239.791,E2 -28239.791} C_VEL
LIN {X 0,Y 121.872,Z 379.585,A -85,B 0,C 180,E1 -28243.238,E2 -28243.238} C_VEL
LIN {X 0,Y 121.372,Z 380.04,A -85,B 0,C 180,E1 -28246.604,E2 -28246.604} C_VEL
LIN {X 0,Y 120.758,Z 380.533,A -85,B 0,C 180,E1 -28248.243,E2 -28248.243} C_VEL
LIN {X 0,Y 113.89,Z 383.632,A -85,B 0,C 180,E1 -28250.862,E2 -28250.862} C_VEL
LIN {X 0,Y 105.97,Z 386.556,A -85,B 0,C 180,E1 -28254.144,E2 -28254.144} C_VEL
LIN {X 0,Y 95.201,Z 389.367,A -85,B 0,C 180,E1 -28259.995,E2 -28259.995} C_VEL
LIN {X 0,Y 88.881,Z 390.372,A -85,B 0,C 180,E1 -28264.53,E2 -28264.53} C_VEL
LIN {X 0,Y 83.257,Z 390.687,A -85,B 0,C 180,E1 -28269.714,E2 -28269.714} C_VEL
LIN {X 0,Y 78.466,Z 390.363,A -85,B 0,C 180,E1 -28275.581,E2 -28275.581} C_VEL
LIN {X 0,Y 74.569,Z 389.406,A -85,B 0,C 180,E1 -28282.14,E2 -28282.14} C_VEL
LIN {X 0,Y 70.668,Z 386.728,A -85,B 0,C 180,E1 -28292.849,E2 -28292.849} C_VEL
LIN {X 0,Y 69.174,Z 382.364,A -85,B 0,C 180,E1 -28304.67,E2 -28304.67} C_VEL
LIN {X 0,Y 69.943,Z 376.778,A -85,B 0,C 180,E1 -28315.45,E2 -28315.45} C_VEL
LIN {X 0,Y 71.766,Z 371.137,A -85,B 0,C 180,E1 -28323.62,E2 -28323.62} C_VEL
LIN {X 0,Y 75.067,Z 363.049,A -85,B 0,C 180,E1 -28332.381,E2 -28332.381} C_VEL
LIN {X 0,Y 78.971,Z 354.372,A -85,B 0,C 180,E1 -28339.306,E2 -28339.306} C_VEL
LIN {X 0,Y 83.512,Z 344.328,A -85,B 0,C 180,E1 -28345.173,E2 -28345.173} C_VEL
LIN {X 0,Y 85.377,Z 339.674,A -85,B 0,C 180,E1 -28347.394,E2 -28347.394} C_VEL
LIN {X 0,Y 85.006,Z 335.236,A -85,B 0,C 180,E1 -28350.037,E2 -28350.037} C_VEL
LIN {X 0,Y 83.729,Z 331.055,A -85,B 0,C 180,E1 -28352.802,E2 -28352.802} C_VEL
LIN {X 0,Y 82.56,Z 328.4,A -85,B 0,C 180,E1 -28354.695,E2 -28354.695} C_VEL
LIN {X 0,Y 77.274,Z 317.74,A -85,B 0,C 180,E1 -28362.713,E2 -28362.713} C_VEL
LIN {X 0,Y 74.734,Z 311.7,A -85,B 0,C 180,E1 -28367.317,E2 -28367.317} C_VEL
LIN {X 0,Y 73.006,Z 308.308,A -85,B 0,C 180,E1 -28370.277,E2 -28370.277} C_VEL
LIN {X 0,Y 68.157,Z 300.15,A -85,B 0,C 180,E1 -28378.802,E2 -28378.802} C_VEL
LIN {X 0,Y 65.822,Z 297.488,A -85,B 0,C 180,E1 -28383.183,E2 -28383.183} C_VEL
LIN {X 0,Y 65.256,Z 295.356,A -85,B 0,C 180,E1 -28385.135,E2 -28385.135} C_VEL
LIN {X 0,Y 65.249,Z 295.317,A -85,B 0,C 180,E1 -28391.076,E2 -28391.076} C_VEL
LIN {X 0,Y 65.264,Z 295.356,A -85,B 0,C 180,E1 -28399.76,E2 -28399.76} C_VEL
LIN {X 0,Y 65.256,Z 295.305,A -85,B 0,C 180,E1 -28409.496,E2 -28409.496} C_VEL
LIN {X 0,Y 65.242,Z 295.34,A -85,B 0,C 180,E1 -28414.485,E2 -28414.485} C_VEL
LIN {X 0,Y 65.622,Z 295.272,A -85,B 0,C 180,E1 -28424.553,E2 -28424.553} C_VEL
LIN {X 0,Y 65.745,Z 295.244,A -85,B 0,C 180,E1 -28427.663,E2 -28427.663} C_VEL
LIN {X 0,Y 66.492,Z 295.19,A -85,B 0,C 180,E1 -28440.007,E2 -28440.007} C_VEL
LIN {X 0,Y 65.862,Z 295.438,A -85,B 0,C 180,E1 -28450.964,E2 -28450.964} C_VEL
LIN {X 0,Y 66.775,Z 298.243,A -85,B 0,C 180,E1 -28453.585,E2 -28453.585} C_VEL
LIN {X 0,Y 68.107,Z 299.885,A -85,B 0,C 180,E1 -28455.984,E2 -28455.984} C_VEL
LIN {X 0,Y 72.024,Z 306.835,A -85,B 0,C 180,E1 -28462.981,E2 -28462.981} C_VEL
LIN {X 0,Y 75.687,Z 314.364,A -85,B 0,C 180,E1 -28469.183,E2 -28469.183} C_VEL
LIN {X 0,Y 77.701,Z 319.702,A -85,B 0,C 180,E1 -28472.874,E2 -28472.874} C_VEL
LIN {X 0,Y 78.77,Z 326.339,A -85,B 0,C 180,E1 -28476.583,E2 -28476.583} C_VEL
LIN {X 0,Y 77.636,Z 337.614,A -85,B 0,C 180,E1 -28482.053,E2 -28482.053} C_VEL
LIN {X 0,Y 76.459,Z 346.766,A -85,B 0,C 180,E1 -28487.345,E2 -28487.345} C_VEL
LIN {X 0,Y 75.732,Z 350.186,A -85,B 0,C 180,E1 -28489.488,E2 -28489.488} C_VEL
LIN {X 0,Y 71.391,Z 359.265,A -85,B 0,C 180,E1 -28495.525,E2 -28495.525} C_VEL
LIN {X 0,Y 67.216,Z 368.057,A -85,B 0,C 180,E1 -28503.616,E2 -28503.616} C_VEL
LIN {X 0,Y 64.434,Z 375.157,A -85,B 0,C 180,E1 -28512.545,E2 -28512.545} C_VEL
LIN {X 0,Y 63.026,Z 381.646,A -85,B 0,C 180,E1 -28523.597,E2 -28523.597} C_VEL
LIN {X 0,Y 63.032,Z 384.584,A -85,B 0,C 180,E1 -28529.999,E2 -28529.999} C_VEL
LIN {X 0,Y 63.103,Z 386.983,A -85,B 0,C 180,E1 -28536.393,E2 -28536.393} C_VEL
LIN {X 0,Y 64.732,Z 390.466,A -85,B 0,C 180,E1 -28549.007,E2 -28549.007} C_VEL
LIN {X 0,Y 69.138,Z 392.443,A -85,B 0,C 180,E1 -28560.546,E2 -28560.546} C_VEL
LIN {X 0,Y 76.283,Z 393.101,A -85,B 0,C 180,E1 -28570.157,E2 -28570.157} C_VEL
LIN {X 0,Y 85.246,Z 392.399,A -85,B 0,C 180,E1 -28577.899,E2 -28577.899} C_VEL
LIN {X 0,Y 95.444,Z 390.306,A -85,B 0,C 180,E1 -28584.091,E2 -28584.091} C_VEL
LIN {X 0,Y 100.953,Z 388.739,A -85,B 0,C 180,E1 -28586.654,E2 -28586.654} C_VEL
LIN {X 0,Y 112.637,Z 384.484,A -85,B 0,C 180,E1 -28590.869,E2 -28590.869} C_VEL
LIN {X 0,Y 114.405,Z 383.265,A -85,B 0,C 180,E1 -28594.527,E2 -28594.527} C_VEL
LIN {X 0,Y 115.404,Z 382.488,A -85,B 0,C 180,E1 -28598.564,E2 -28598.564} C_VEL
LIN {X 0,Y 115.418,Z 382.41,A -85,B 0,C 180,E1 -28602.27,E2 -28602.27} C_VEL
LIN {X 0,Y 114.906,Z 382.741,A -85,B 0,C 180,E1 -28605.835,E2 -28605.835} C_VEL
LIN {X 0,Y 111.75,Z 384.028,A -85,B 0,C 180,E1 -28607.28,E2 -28607.28} C_VEL
LIN {X 0,Y 99.779,Z 387.943,A -85,B 0,C 180,E1 -28611.897,E2 -28611.897} C_VEL
LIN {X 0,Y 91.574,Z 389.737,A -85,B 0,C 180,E1 -28616.089,E2 -28616.089} C_VEL
LIN {X 0,Y 84.342,Z 390.683,A -85,B 0,C 180,E1 -28620.82,E2 -28620.82} C_VEL
LIN {X 0,Y 77.799,Z 390.918,A -85,B 0,C 180,E1 -28626.455,E2 -28626.455} C_VEL
LIN {X 0,Y 72.156,Z 390.367,A -85,B 0,C 180,E1 -28633.102,E2 -28633.102} C_VEL
LIN {X 0,Y 67.638,Z 389.06,A -85,B 0,C 180,E1 -28640.753,E2 -28640.753} C_VEL
LIN {X 0,Y 64.386,Z 387.025,A -85,B 0,C 180,E1 -28649.168,E2 -28649.168} C_VEL
LIN {X 0,Y 62.539,Z 384.224,A -85,B 0,C 180,E1 -28658.13,E2 -28658.13} C_VEL
LIN {X 0,Y 62.226,Z 379.355,A -85,B 0,C 180,E1 -28669.891,E2 -28669.891} C_VEL
LIN {X 0,Y 63.463,Z 374.389,A -85,B 0,C 180,E1 -28679.055,E2 -28679.055} C_VEL
LIN {X 0,Y 65.79,Z 368.179,A -85,B 0,C 180,E1 -28687.862,E2 -28687.862} C_VEL
LIN {X 0,Y 69.727,Z 359.579,A -85,B 0,C 180,E1 -28696.893,E2 -28696.893} C_VEL
LIN {X 0,Y 74.204,Z 350.352,A -85,B 0,C 180,E1 -28703.884,E2 -28703.884} C_VEL
LIN {X 0,Y 78.391,Z 341.435,A -85,B 0,C 180,E1 -28708.855,E2 -28708.855} C_VEL
LIN {X 0,Y 78.917,Z 339.321,A -85,B 0,C 180,E1 -28710.001,E2 -28710.001} C_VEL
LIN {X 0,Y 79.458,Z 330.282,A -85,B 0,C 180,E1 -28715.075,E2 -28715.075} C_VEL
LIN {X 0,Y 79.452,Z 324.571,A -85,B 0,C 180,E1 -28718.1,E2 -28718.1} C_VEL
LIN {X 0,Y 78.134,Z 319.869,A -85,B 0,C 180,E1 -28721.16,E2 -28721.16} C_VEL
LIN {X 0,Y 77.274,Z 317.74,A -85,B 0,C 180,E1 -28722.713,E2 -28722.713} C_VEL
LIN {X 0,Y 75.152,Z 314.169,A -85,B 0,C 180,E1 -28725.865,E2 -28725.865} C_VEL
LIN {X 0,Y 72.342,Z 311.441,A -85,B 0,C 180,E1 -28729.342,E2 -28729.342} C_VEL
LIN {X 0,Y 62.985,Z 304.36,A -85,B 0,C 180,E1 -28743.427,E2 -28743.427} C_VEL
LIN {X 0,Y 61.735,Z 301.532,A -85,B 0,C 180,E1 -28747.179,E2 -28747.179} C_VEL
LIN {X 0,Y 58.688,Z 298.331,A -85,B 0,C 180,E1 -28756.243,E2 -28756.243} C_VEL
LIN {X 0,Y 58.23,Z 296.232,A -85,B 0,C 180,E1 -28759.686,E2 -28759.686} C_VEL
LIN {X 0,Y 58.167,Z 296.189,A -85,B 0,C 180,E1 -28767.754,E2 -28767.754} C_VEL
LIN {X 0,Y 58.152,Z 296.193,A -85,B 0,C 180,E1 -28771.1,E2 -28771.1} C_VEL
LIN {X 0,Y 58.514,Z 296.16,A -85,B 0,C 180,E1 -28783.917,E2 -28783.917} C_VEL
LIN {X 0,Y 58.791,Z 296.14,A -85,B 0,C 180,E1 -28793.143,E2 -28793.143} C_VEL
LIN {X 0,Y 59.257,Z 296.312,A -85,B 0,C 180,E1 -28798.734,E2 -28798.734} C_VEL
LIN {X 0,Y 59.67,Z 297.618,A -85,B 0,C 180,E1 -28800.852,E2 -28800.852} C_VEL
LIN {X 0,Y 60.248,Z 299.261,A -85,B 0,C 180,E1 -28803.352,E2 -28803.352} C_VEL
LIN {X 0,Y 62.611,Z 302.403,A -85,B 0,C 180,E1 -28809.701,E2 -28809.701} C_VEL
LIN {X 0,Y 64.534,Z 305.906,A -85,B 0,C 180,E1 -28814.49,E2 -28814.49} C_VEL
LIN {X 0,Y 67.604,Z 312.014,A -85,B 0,C 180,E1 -28821.345,E2 -28821.345} C_VEL
LIN {X 0,Y 70.841,Z 319.505,A -85,B 0,C 180,E1 -28828.122,E2 -28828.122} C_VEL
LIN {X 0,Y 72.166,Z 324.108,A -85,B 0,C 180,E1 -28831.572,E2 -28831.572} C_VEL
LIN {X 0,Y 72.669,Z 327.566,A -85,B 0,C 180,E1 -28833.794,E2 -28833.794} C_VEL
LIN {X 0,Y 71.4,Z 337.766,A -85,B 0,C 180,E1 -28839.294,E2 -28839.294} C_VEL
LIN {X 0,Y 69.887,Z 347.221,A -85,B 0,C 180,E1 -28845.257,E2 -28845.257} C_VEL
LIN {X 0,Y 68.964,Z 350.621,A -85,B 0,C 180,E1 -28847.535,E2 -28847.535} C_VEL
LIN {X 0,Y 63.947,Z 360.313,A -85,B 0,C 180,E1 -28854.76,E2 -28854.76} C_VEL
LIN {X 0,Y 59.7,Z 368.885,A -85,B 0,C 180,E1 -28863.802,E2 -28863.802} C_VEL
LIN {X 0,Y 57.01,Z 375.778,A -85,B 0,C 180,E1 -28873.896,E2 -28873.896} C_VEL
LIN {X 0,Y 56.019,Z 380.425,A -85,B 0,C 180,E1 -28882.792,E2 -28882.792} C_VEL
LIN {X 0,Y 55.996,Z 383.535,A -85,B 0,C 180,E1 -28889.999,E2 -28889.999} C_VEL
LIN {X 0,Y 56.115,Z 386.039,A -85,B 0,C 180,E1 -28897.194,E2 -28897.194} C_VEL
LIN {X 0,Y 58.085,Z 389.73,A -85,B 0,C 180,E1 -28911.282,E2 -28911.282} C_VEL
LIN {X 0,Y 63.119,Z 391.979,A -85,B 0,C 180,E1 -28923.828,E2 -28923.828} C_VEL
LIN {X 0,Y 70.997,Z 392.845,A -85,B 0,C 180,E1 -28933.86,E2 -28933.86} C_VEL
LIN {X 0,Y 80.65,Z 392.379,A -85,B 0,C 180,E1 -28941.651,E2 -28941.651} C_VEL
LIN {X 0,Y 91.463,Z 390.583,A -85,B 0,C 180,E1 -28947.695,E2 -28947.695} C_VEL
LIN {X 0,Y 103.253,Z 387.358,A -85,B 0,C 180,E1 -28952.23,E2 -28952.23} C_VEL
LIN {X 0,Y 106.309,Z 386.332,A -85,B 0,C 180,E1 -28953.183,E2 -28953.183} C_VEL
LIN {X 0,Y 107.98,Z 385.521,A -85,B 0,C 180,E1 -28955.669,E2 -28955.669} C_VEL
LIN {X 0,Y 108.416,Z 385.245,A -85,B 0,C 180,E1 -28957.107,E2 -28957.107} C_VEL
LIN {X 0,Y 108.736,Z 384.952,A -85,B 0,C 180,E1 -28961.141,E2 -28961.141} C_VEL
LIN {X 0,Y 108.595,Z 384.999,A -85,B 0,C 180,E1 -28963.064,E2 -28963.064} C_VEL
LIN {X 0,Y 106.415,Z 385.749,A -85,B 0,C 180,E1 -28964.678,E2 -28964.678} C_VEL
LIN {X 0,Y 98.049,Z 388.16,A -85,B 0,C 180,E1 -28967.577,E2 -28967.577} C_VEL
LIN {X 0,Y 90.162,Z 389.809,A -85,B 0,C 180,E1 -28971.026,E2 -28971.026} C_VEL
LIN {X 0,Y 82.716,Z 390.825,A -85,B 0,C 180,E1 -28975.12,E2 -28975.12} C_VEL
LIN {X 0,Y 75.815,Z 391.148,A -85,B 0,C 180,E1 -28979.994,E2 -28979.994} C_VEL
LIN {X 0,Y 69.621,Z 390.848,A -85,B 0,C 180,E1 -28985.787,E2 -28985.787} C_VEL
LIN {X 0,Y 64.292,Z 389.907,A -85,B 0,C 180,E1 -28992.621,E2 -28992.621} C_VEL
LIN {X 0,Y 58.35,Z 387.234,A -85,B 0,C 180,E1 -29004.92,E2 -29004.92} C_VEL
LIN {X 0,Y 55.947,Z 384.546,A -85,B 0,C 180,E1 -29014.407,E2 -29014.407} C_VEL
LIN {X 0,Y 55.032,Z 380.683,A -85,B 0,C 180,E1 -29025.364,E2 -29025.364} C_VEL
LIN {X 0,Y 56.052,Z 374.997,A -85,B 0,C 180,E1 -29037.802,E2 -29037.802} C_VEL
LIN {X 0,Y 58.133,Z 369.475,A -85,B 0,C 180,E1 -29046.916,E2 -29046.916} C_VEL
LIN {X 0,Y 62,Z 361.313,A -85,B 0,C 180,E1 -29056.898,E2 -29056.898} C_VEL
LIN {X 0,Y 67.169,Z 351.394,A -85,B 0,C 180,E1 -29065.421,E2 -29065.421} C_VEL
LIN {X 0,Y 72.131,Z 341.447,A -85,B 0,C 180,E1 -29071.397,E2 -29071.397} C_VEL
LIN {X 0,Y 72.993,Z 334.83,A -85,B 0,C 180,E1 -29075.526,E2 -29075.526} C_VEL
LIN {X 0,Y 73.386,Z 327.267,A -85,B 0,C 180,E1 -29080.013,E2 -29080.013} C_VEL
LIN {X 0,Y 72.215,Z 322.901,A -85,B 0,C 180,E1 -29083.323,E2 -29083.323} C_VEL
LIN {X 0,Y 69.899,Z 316.711,A -85,B 0,C 180,E1 -29088.557,E2 -29088.557} C_VEL
LIN {X 0,Y 67.596,Z 312.19,A -85,B 0,C 180,E1 -29093.151,E2 -29093.151} C_VEL
LIN {X 0,Y 64.696,Z 306.59,A -85,B 0,C 180,E1 -29099.668,E2 -29099.668} C_VEL
LIN {X 0,Y 62.985,Z 304.36,A -85,B 0,C 180,E1 -29103.427,E2 -29103.427} C_VEL
LIN {X 0,Y 60.809,Z 302.543,A -85,B 0,C 180,E1 -29108.25,E2 -29108.25} C_VEL
LIN {X 0,Y 58.586,Z 301.77,A -85,B 0,C 180,E1 -29113.517,E2 -29113.517} C_VEL
LIN {X 0,Y 53.915,Z 301.998,A -85,B 0,C 180,E1 -29133.79,E2 -29133.79} C_VEL
LIN {X 0,Y 54.286,Z 301.814,A -85,B 0,C 180,E1 -29145.003,E2 -29145.003} C_VEL
LIN {X 0,Y 56.35,Z 302.737,A -85,B 0,C 180,E1 -29156.166,E2 -29156.166} C_VEL
LIN {X 0,Y 58.805,Z 307.776,A -85,B 0,C 180,E1 -29166.872,E2 -29166.872} C_VEL
LIN {X 0,Y 60.849,Z 312.138,A -85,B 0,C 180,E1 -29173.364,E2 -29173.364} C_VEL
LIN {X 0,Y 63.045,Z 317.055,A -85,B 0,C 180,E1 -29179.545,E2 -29179.545} C_VEL
LIN {X 0,Y 65.79,Z 324.442,A -85,B 0,C 180,E1 -29187.009,E2 -29187.009} C_VEL
LIN {X 0,Y 66.547,Z 328.364,A -85,B 0,C 180,E1 -29190.117,E2 -29190.117} C_VEL
LIN {X 0,Y 66.474,Z 331.635,A -85,B 0,C 180,E1 -29192.242,E2 -29192.242} C_VEL
LIN {X 0,Y 64.482,Z 342.531,A -85,B 0,C 180,E1 -29199.053,E2 -29199.053} C_VEL
LIN {X 0,Y 62.799,Z 349.993,A -85,B 0,C 180,E1 -29204.486,E2 -29204.486} C_VEL
LIN {X 0,Y 57.402,Z 359.777,A -85,B 0,C 180,E1 -29212.253,E2 -29212.253} C_VEL
LIN {X 0,Y 52.792,Z 368.398,A -85,B 0,C 180,E1 -29222.228,E2 -29222.228} C_VEL
LIN {X 0,Y 49.89,Z 375.331,A -85,B 0,C 180,E1 -29233.635,E2 -29233.635} C_VEL
LIN {X 0,Y 48.908,Z 380.832,A -85,B 0,C 180,E1 -29245.879,E2 -29245.879} C_VEL
LIN {X 0,Y 49.034,Z 383.756,A -85,B 0,C 180,E1 -29254.108,E2 -29254.108} C_VEL
LIN {X 0,Y 49.827,Z 387.178,A -85,B 0,C 180,E1 -29266.384,E2 -29266.384} C_VEL
LIN {X 0,Y 54.026,Z 390.356,A -85,B 0,C 180,E1 -29281.353,E2 -29281.353} C_VEL
LIN {X 0,Y 61.477,Z 392.159,A -85,B 0,C 180,E1 -29293.306,E2 -29293.306} C_VEL
LIN {X 0,Y 71.06,Z 392.629,A -85,B 0,C 180,E1 -29302.297,E2 -29302.297} C_VEL
LIN {X 0,Y 82.028,Z 391.729,A -85,B 0,C 180,E1 -29308.954,E2 -29308.954} C_VEL
LIN {X 0,Y 93.916,Z 389.511,A -85,B 0,C 180,E1 -29313.892,E2 -29313.892} C_VEL
LIN {X 0,Y 100.151,Z 387.88,A -85,B 0,C 180,E1 -29315.815,E2 -29315.815} C_VEL
LIN {X 0,Y 101.811,Z 387.197,A -85,B 0,C 180,E1 -29319.804,E2 -29319.804} C_VEL
LIN {X 0,Y 101.321,Z 387.29,A -85,B 0,C 180,E1 -29321.807,E2 -29321.807} C_VEL
LIN {X 0,Y 95.181,Z 388.797,A -85,B 0,C 180,E1 -29323.714,E2 -29323.714} C_VEL
LIN {X 0,Y 86.525,Z 390.378,A -85,B 0,C 180,E1 -29327.078,E2 -29327.078} C_VEL
LIN {X 0,Y 78.223,Z 391.208,A -85,B 0,C 180,E1 -29331.214,E2 -29331.214} C_VEL
LIN {X 0,Y 70.418,Z 391.348,A -85,B 0,C 180,E1 -29336.376,E2 -29336.376} C_VEL
LIN {X 0,Y 63.325,Z 390.759,A -85,B 0,C 180,E1 -29342.789,E2 -29342.789} C_VEL
LIN {X 0,Y 54.936,Z 388.551,A -85,B 0,C 180,E1 -29354.815,E2 -29354.815} C_VEL
LIN {X 0,Y 51.032,Z 386.292,A -85,B 0,C 180,E1 -29364.393,E2 -29364.393} C_VEL
LIN {X 0,Y 48.258,Z 382.024,A -85,B 0,C 180,E1 -29379.055,E2 -29379.055} C_VEL
LIN {X 0,Y 48.482,Z 376.207,A -85,B 0,C 180,E1 -29394.563,E2 -29394.563} C_VEL
LIN {X 0,Y 50.374,Z 370.883,A -85,B 0,C 180,E1 -29405.259,E2 -29405.259} C_VEL
LIN {X 0,Y 54.206,Z 363.112,A -85,B 0,C 180,E1 -29416.778,E2 -29416.778} C_VEL
LIN {X 0,Y 58.995,Z 354.387,A -85,B 0,C 180,E1 -29425.731,E2 -29425.731} C_VEL
LIN {X 0,Y 64.835,Z 343.809,A -85,B 0,C 180,E1 -29433.108,E2 -29433.108} C_VEL
LIN {X 0,Y 66.05,Z 341.241,A -85,B 0,C 180,E1 -29434.578,E2 -29434.578} C_VEL
LIN {X 0,Y 67.254,Z 331.876,A -85,B 0,C 180,E1 -29440.951,E2 -29440.951} C_VEL
LIN {X 0,Y 67.375,Z 330.223,A -85,B 0,C 180,E1 -29442.042,E2 -29442.042} C_VEL
LIN {X 0,Y 66.536,Z 326.536,A -85,B 0,C 180,E1 -29445.165,E2 -29445.165} C_VEL
LIN {X 0,Y 64.399,Z 320.207,A -85,B 0,C 180,E1 -29451.312,E2 -29451.312} C_VEL
LIN {X 0,Y 62.275,Z 315.584,A -85,B 0,C 180,E1 -29456.835,E2 -29456.835} C_VEL
